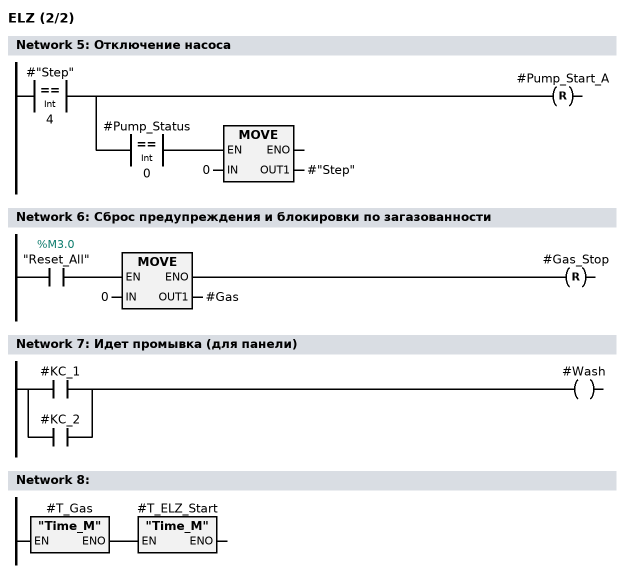
   RUNG wire#powerrail
      { S7_Templates := "SrcType := Int" } EQ_Contact(in1 := #"Step", in2 := 4)
      wire#w1
      R_Coil( #Pump_Start_A )
   END_RUNG
   RUNG wire#w1
      { S7_Templates := "SrcType := Int" } EQ_Contact(in1 := #Pump_Status, in2 := 0)
      Move(in := 0, out1 => #"Step")
   END_RUNG
   // the same network as SCL:
   #_w1 := #"Step" = 4;
   IF #_w1 THEN #Pump_Start_A := FALSE; END_IF;
   IF #_w1 AND (#Pump_Status = 0) THEN #"Step" := 0; END_IF;
END_REGION

REGION Network 6: Сброс предупреждения и блокировки по загазованности
   RUNG wire#powerrail
      Contact( "Reset_All" )
      Move(in := 0, out1 => #Gas)
      R_Coil( #Gas_Stop )
   END_RUNG
   // the same network as SCL:
   IF "Reset_All" THEN
       #Gas := 0;
       #Gas_Stop := FALSE;
   END_IF;
END_REGION

REGION Network 7: Идет промывка (для панели)
   RUNG wire#powerrail
      Contact( #KC_1 )
      wire#w1
      Coil( #Wash )
   END_RUNG
   RUNG wire#powerrail
      Contact( #KC_2 )
   END_RUNG wire#w1
   // the same network as SCL:
   #Wash := #KC_1 OR #KC_2;
END_REGION

REGION Network 8
   RUNG wire#powerrail
      #T_Gas()
      #T_ELZ_Start()
   END_RUNG
   // the same network as SCL:
   #T_Gas(ENO => #_w1);   // "Time_M"
   IF #_w1 THEN
       #T_ELZ_Start();   // "Time_M"
   END_IF;
END_REGION
END_FUNCTION_BLOCK

FUNCTION_BLOCK "Time_M"   // FB92, LAD
{ S7_Optimized_Access := 'FALSE' }
VERSION : 0.1
// stored: AutoNumber false, IsIECCheckEnabled false, SetENOAutomatically false, UDAEnableTagReadback false
   VAR DB_SPECIFIC
      SP_M { S7_SetPoint := 'True'} : Int;
      SP_S { S7_SetPoint := 'True'} : Int := 30;
      Now_M : Int;
      Now_S : Int;
      Rev_M : Int;
      Rev_S : Int;
      Progress : Real;
      Start : Bool;
      "Exit" : Bool;
      Pause : Bool;
      Reset : Bool;
   END_VAR
   VAR_TEMP
      Full_SP_S : Int;
      Full_Now_S : Int;
      Full_Delta_S : Int;
   END_VAR
   VAR_TEMP   // added for the SCL form of the ladder/FBD networks
      _w1 : Bool;
   END_VAR
BEGIN

REGION Network 1: Подсчёт времени
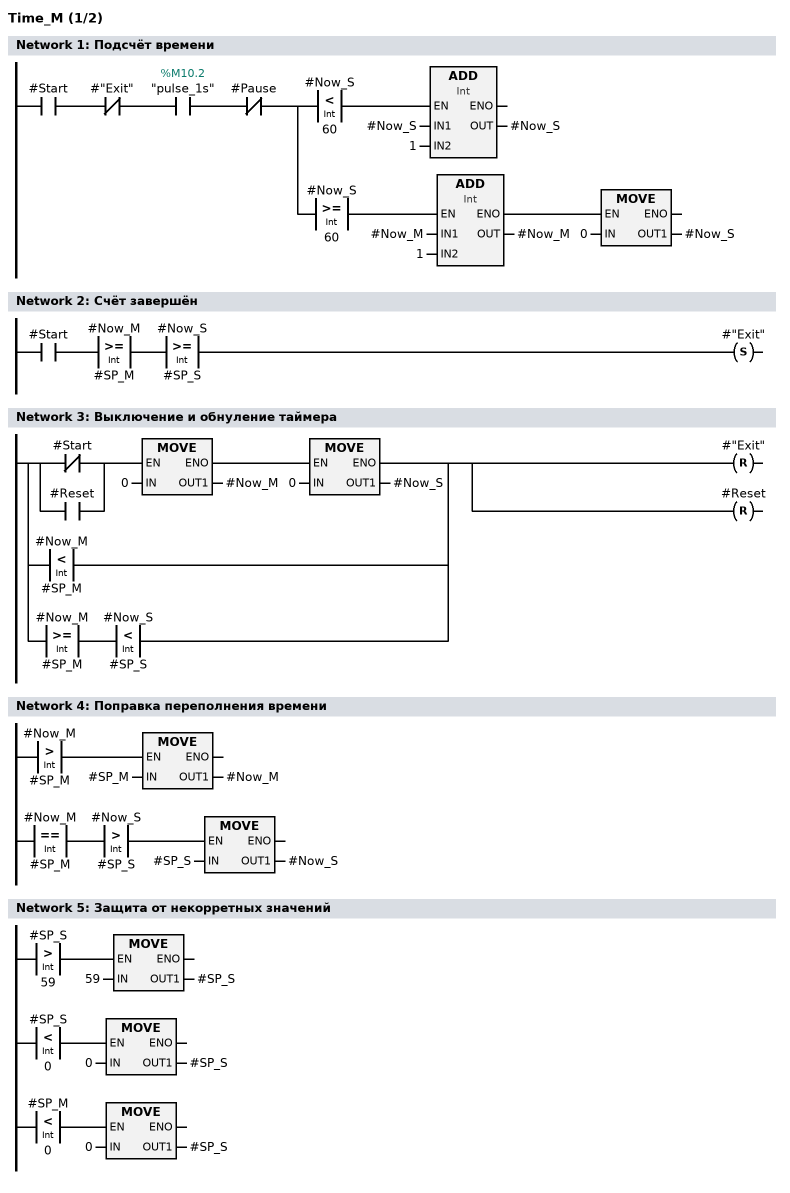
   RUNG wire#powerrail
      Contact( #Start )
      I_Contact( #"Exit" )
      Contact( "pulse_1s" )
      I_Contact( #Pause )
      wire#w1
      { S7_Templates := "SrcType := Int" } LT_Contact(in1 := #Now_S, in2 := 60)
      { S7_Templates := "SrcType := Int"; S7_GenerateENO := "TRUE" } Add(in1 := #Now_S, in2 := 1, out => #Now_S)
   END_RUNG
   RUNG wire#w1
      { S7_Templates := "SrcType := Int" } GE_Contact(in1 := #Now_S, in2 := 60)
      { S7_Templates := "SrcType := Int"; S7_GenerateENO := "TRUE" } Add(in1 := #Now_M, in2 := 1, out => #Now_M)
      { S7_GenerateENO := "TRUE" } Move(in := 0, out1 => #Now_S)
   END_RUNG
   // the same network as SCL:
   // ENO of a box is taken as its EN; it also drops when the box reports an error
   #_w1 := #Start AND NOT #"Exit" AND "pulse_1s" AND NOT #Pause;
   IF #_w1 AND (#Now_S < 60) THEN #Now_S := #Now_S + 1; END_IF;
   IF #_w1 AND (#Now_S >= 60) THEN
       #Now_M := #Now_M + 1;
       #Now_S := 0;
   END_IF;
END_REGION

REGION Network 2: Счёт завершён
   RUNG wire#powerrail
      Contact( #Start )
      { S7_Templates := "SrcType := Int" } GE_Contact(in1 := #Now_M, in2 := #SP_M)
      { S7_Templates := "SrcType := Int" } GE_Contact(in1 := #Now_S, in2 := #SP_S)
      S_Coil( #"Exit" )
   END_RUNG
   // the same network as SCL:
   IF #Start AND (#Now_M >= #SP_M) AND (#Now_S >= #SP_S) THEN #"Exit" := TRUE; END_IF;
END_REGION

REGION Network 3: Выключение и обнуление таймера
   RUNG wire#powerrail
      I_Contact( #Start )
      wire#w1
      { S7_GenerateENO := "TRUE" } Move(in := 0, out1 => #Now_M)
      { S7_GenerateENO := "TRUE" } Move(in := 0, out1 => #Now_S)
      wire#w2
      R_Coil( #"Exit" )
   END_RUNG
   RUNG wire#powerrail
      Contact( #Reset )
   END_RUNG wire#w1
   RUNG wire#powerrail
      { S7_Templates := "SrcType := Int" } LT_Contact(in1 := #Now_M, in2 := #SP_M)
   END_RUNG wire#w2
   RUNG wire#powerrail
      { S7_Templates := "SrcType := Int" } GE_Contact(in1 := #Now_M, in2 := #SP_M)
      { S7_Templates := "SrcType := Int" } LT_Contact(in1 := #Now_S, in2 := #SP_S)
   END_RUNG wire#w2
   RUNG wire#w2
      R_Coil( #Reset )
   END_RUNG
   // the same network as SCL:
   // ENO of a box is taken as its EN; it also drops when the box reports an error
   #_w1 := NOT #Start OR #Reset;
   IF #_w1 THEN
       #Now_M := 0;
       #Now_S := 0;
   END_IF;
   IF #_w1 OR (#Now_M < #SP_M) OR ((#Now_M >= #SP_M) AND (#Now_S < #SP_S)) THEN
       #"Exit" := FALSE;
       #Reset := FALSE;
   END_IF;
END_REGION

REGION Network 4: Поправка переполнения времени
   RUNG wire#powerrail
      { S7_Templates := "SrcType := Int" } GT_Contact(in1 := #Now_M, in2 := #SP_M)
      { S7_GenerateENO := "TRUE" } Move(in := #SP_M, out1 => #Now_M)
   END_RUNG
   RUNG wire#powerrail
      { S7_Templates := "SrcType := Int" } EQ_Contact(in1 := #Now_M, in2 := #SP_M)
      { S7_Templates := "SrcType := Int" } GT_Contact(in1 := #Now_S, in2 := #SP_S)
      { S7_GenerateENO := "TRUE" } Move(in := #SP_S, out1 => #Now_S)
   END_RUNG
   // the same network as SCL:
   IF #Now_M > #SP_M THEN #Now_M := #SP_M; END_IF;
   IF (#Now_M = #SP_M) AND (#Now_S > #SP_S) THEN #Now_S := #SP_S; END_IF;
END_REGION

REGION Network 5: Защита от некорретных значений
   RUNG wire#powerrail
      { S7_Templates := "SrcType := Int" } GT_Contact(in1 := #SP_S, in2 := 59)
      { S7_GenerateENO := "TRUE" } Move(in := 59, out1 => #SP_S)
   END_RUNG
   RUNG wire#powerrail
      { S7_Templates := "SrcType := Int" } LT_Contact(in1 := #SP_S, in2 := 0)
      { S7_GenerateENO := "TRUE" } Move(in := 0, out1 => #SP_S)
   END_RUNG
   RUNG wire#powerrail
      { S7_Templates := "SrcType := Int" } LT_Contact(in1 := #SP_M, in2 := 0)
      { S7_GenerateENO := "TRUE" } Move(in := 0, out1 => #SP_S)
   END_RUNG
   // the same network as SCL:
   IF #SP_S > 59 THEN #SP_S := 59; END_IF;
   IF #SP_S < 0 THEN #SP_S := 0; END_IF;
   IF #SP_M < 0 THEN #SP_S := 0; END_IF;
END_REGION

REGION Network 6: Обратный отсчёт
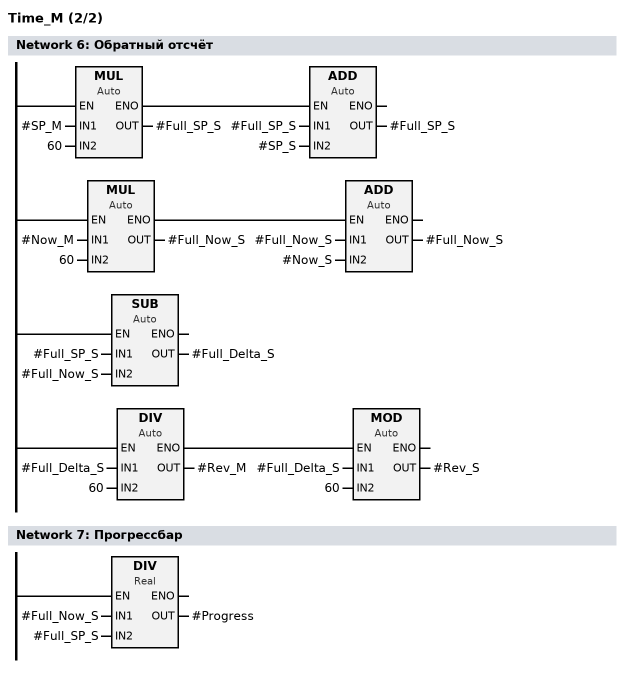
   RUNG wire#powerrail
      Mul(in1 := #SP_M, in2 := 60, out => #Full_SP_S)
      Add(in1 := #Full_SP_S, in2 := #SP_S, out => #Full_SP_S)
   END_RUNG
   RUNG wire#powerrail
      Mul(in1 := #Now_M, in2 := 60, out => #Full_Now_S)
      Add(in1 := #Full_Now_S, in2 := #Now_S, out => #Full_Now_S)
   END_RUNG
   RUNG wire#powerrail
      Sub(in1 := #Full_SP_S, in2 := #Full_Now_S, out => #Full_Delta_S)
   END_RUNG
   RUNG wire#powerrail
      Div(in1 := #Full_Delta_S, in2 := 60, out => #Rev_M)
      Mod(in1 := #Full_Delta_S, in2 := 60, out => #Rev_S)
   END_RUNG
   // the same network as SCL:
   #Full_SP_S := #SP_M * 60;
   #Full_SP_S := #Full_SP_S + #SP_S;
   #Full_Now_S := #Now_M * 60;
   #Full_Now_S := #Full_Now_S + #Now_S;
   #Full_Delta_S := #Full_SP_S - #Full_Now_S;
   #Rev_M := #Full_Delta_S / 60;
   #Rev_S := #Full_Delta_S MOD 60;
END_REGION

REGION Network 7: Прогрессбар
   RUNG wire#powerrail
      { S7_Templates := "SrcType := Real" } Div(in1 := #Full_Now_S, in2 := #Full_SP_S, out => #Progress)
   END_RUNG
   // the same network as SCL:
   #Progress := #Full_Now_S / #Full_SP_S;
END_REGION
END_FUNCTION_BLOCK

FUNCTION_BLOCK "Lock"   // FB2, LAD
{ S7_Optimized_Access := 'TRUE' }
VERSION : 0.1
// stored: AutoNumber true, IsIECCheckEnabled false, IsRetainMemResEnabled false, MemoryReserve 100, SetENOAutomatically false, UDAEnableTagReadback false
BEGIN

REGION Network 1: Блокировка электролизера
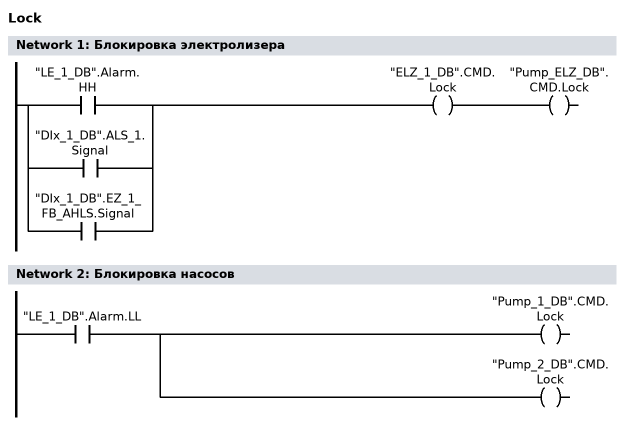
   RUNG wire#powerrail
      Contact( "LE_1_DB".Alarm.HH )
      wire#w1
      Coil( "ELZ_1_DB".CMD.Lock )
      Coil( "Pump_ELZ_DB".CMD.Lock )
   END_RUNG
   RUNG wire#powerrail
      Contact( "DIx_1_DB".ALS_1.Signal )
   END_RUNG wire#w1
   RUNG wire#powerrail
      Contact( "DIx_1_DB".EZ_1_FB_AHLS.Signal )
   END_RUNG wire#w1
   // the same network as SCL:
   "ELZ_1_DB".CMD.Lock := "LE_1_DB".Alarm.HH OR "DIx_1_DB".ALS_1.Signal OR "DIx_1_DB".EZ_1_FB_AHLS.Signal;
   "Pump_ELZ_DB".CMD.Lock := "ELZ_1_DB".CMD.Lock;
END_REGION

REGION Network 2: Блокировка насосов
   RUNG wire#powerrail
      Contact( "LE_1_DB".Alarm.LL )
      wire#w1
      Coil( "Pump_1_DB".CMD.Lock )
   END_RUNG
   RUNG wire#w1
      Coil( "Pump_2_DB".CMD.Lock )
   END_RUNG
   // the same network as SCL:
   "Pump_1_DB".CMD.Lock := "LE_1_DB".Alarm.LL;
   "Pump_2_DB".CMD.Lock := "LE_1_DB".Alarm.LL;
END_REGION
END_FUNCTION_BLOCK

FUNCTION_BLOCK "Line_Control"   // FB5, LAD
{ S7_Optimized_Access := 'FALSE' }
VERSION : 0.1
// stored: AutoNumber false, IsIECCheckEnabled false, SetENOAutomatically false, UDAEnableTagReadback false
   VAR DB_SPECIFIC
      Local : Bool;   // Локальный
      RESET_STAT : Bool;   // Обнуление статистики за неделю
      Line_Settings : Bool;   // Параметры линии
      Line_Alarms : Bool;   // Аварии линии
      Group1_PolyMix_1 : Bool;   // Группа 1 PolyMix 1
      Group1_PolyMix_2 : Bool;   // Группа 1 PolyMix 2
      Group2_PolyMix_1 : Bool;   // Группа 2 PolyMix 1
      Group2_PolyMix_2 : Bool;   // Группа 2 PolyMix 2
      ALLS : Bool;   // Нижний аварийный уровень
      REQ_Z6_BK1 : Bool;   // Запрос открытия задвижки 6 с БК 1
      REQ_Z6_BK2 : Bool;   // Запрос открытия задвижки 6 с БК 2
      REQ_Z5_Start_A : Bool;   // Запрос открытия задвижки 5
      REQ_Z4_Start_A : Bool;   // Запрос открытия задвижки 4
      REQ_Z3_Start_A : Bool;   // Запрос открытия задвижки 3
      REQ_Z2_Start_A : Bool;   // Запрос открытия задвижки 2
      REQ_Z1_Start_A : Bool;   // Запрос открытия задвижки 1
      Line_REQ_Settings : Int;   // Запрос параметров линии
      Line_Now_Settings : Int;   // Параметры линии сейчас
      Line_REQ_Alarms : Int;   // Запрос аварий линии
      Line_Now_Alarms : Int;   // Аварии линии сейчас
      All_Lines : Int := 1;   // Кол-во линий
      All_Pumps : Int := 2;   // Кол-во насосов
      Events : Word;   // События
      pos : Array[0..7] of Bool;   // Вспомогательные переменные
   END_VAR
   VAR
      Line { S7_SetPoint := 'True'} : Array[0..2] of "Block_Line";   // Линии (Block Line)
      Pump { S7_SetPoint := 'True'} : Array[1..2] of "Block_Pump";   // Насосы (Block Pump)
   END_VAR
   VAR DB_SPECIFIC
      Time_DTL : DTL;
   END_VAR
   VAR_TEMP
      summ : Real;
      x1 : Bool;
      x2 : Bool;
   END_VAR
   // Line[1].Flow := 1.0;
   // Line[1].LINE_NUMBER := 1;
   // Line[2].LINE_NUMBER := 2;
   // Line[1..2].Hand := true;
   // Line[0].PID.Settings.Max_out := 1.3;
   // Line[0].PID.Settings.Min_out := 0.7;
   // Line[0].PID.Settings.DeadBand := 0.0;
   // Pump[1].PUMP_NUMBER := 1;
   // Pump[2].PUMP_NUMBER := 2;
   // Pump[1].Line_Main := 1;
   // Pump[2].Line_Main := 2;
   VAR_TEMP   // added for the SCL form of the ladder/FBD networks
      _w1 : Bool;
   END_VAR
BEGIN

REGION Network 1: Вызов функций настроек и аварий линий
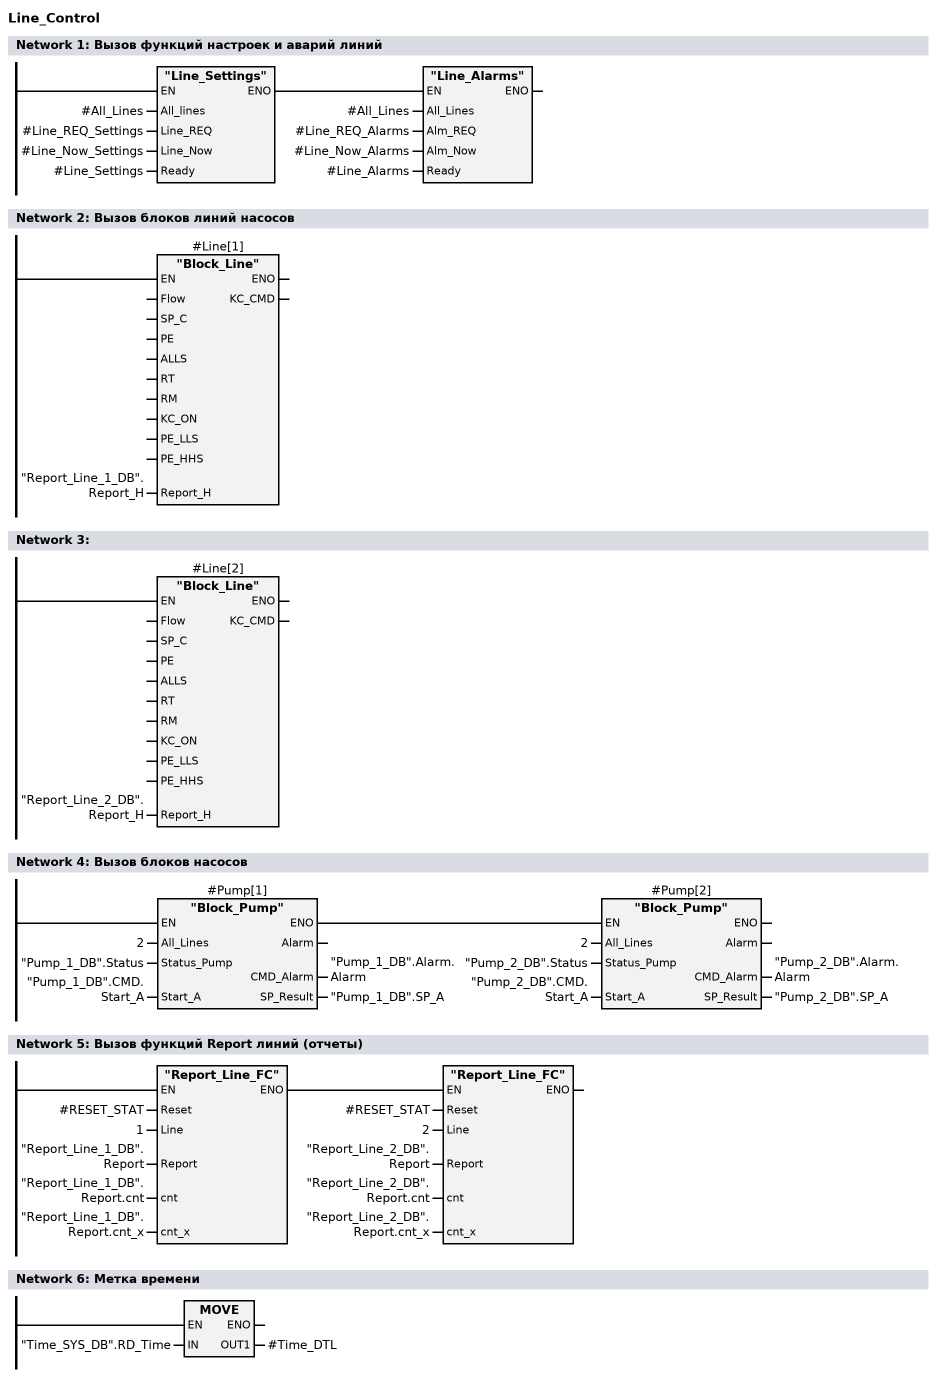
   RUNG wire#powerrail
      "Line_Settings"(All_lines := #All_Lines, Line_REQ := #Line_REQ_Settings, Line_Now := #Line_Now_Settings, Ready := #Line_Settings)
      "Line_Alarms"(All_Lines := #All_Lines, Alm_REQ := #Line_REQ_Alarms, Alm_Now := #Line_Now_Alarms, Ready := #Line_Alarms)
   END_RUNG
   // the same network as SCL:
   "Line_Settings"(All_lines := #All_Lines,
                   Line_REQ := #Line_REQ_Settings,
                   Line_Now := #Line_Now_Settings,
                   Ready := #Line_Settings,
                   ENO => #_w1);
   IF #_w1 THEN
       "Line_Alarms"(All_Lines := #All_Lines,
                     Alm_REQ := #Line_REQ_Alarms,
                     Alm_Now := #Line_Now_Alarms,
                     Ready := #Line_Alarms);
   END_IF;
END_REGION

REGION Network 2: Вызов блоков линий насосов
   RUNG wire#powerrail
      #Line[1](Flow :=, SP_C :=, PE :=, ALLS :=, RT :=, RM :=, KC_ON :=, PE_LLS :=, PE_HHS :=, Report_H := "Report_Line_1_DB".Report_H, KC_CMD =>)
   END_RUNG
   // the same network as SCL:
   #Line[1](Report_H := "Report_Line_1_DB".Report_H);   // "Block_Line"
END_REGION

REGION Network 3
   RUNG wire#powerrail
      #Line[2](Flow :=, SP_C :=, PE :=, ALLS :=, RT :=, RM :=, KC_ON :=, PE_LLS :=, PE_HHS :=, Report_H := "Report_Line_2_DB".Report_H, KC_CMD =>)
   END_RUNG
   // the same network as SCL:
   #Line[2](Report_H := "Report_Line_2_DB".Report_H);   // "Block_Line"
END_REGION

REGION Network 4: Вызов блоков насосов
   RUNG wire#powerrail
      #Pump[1](All_Lines := 2, Status_Pump := "Pump_1_DB".Status, Start_A := "Pump_1_DB".CMD.Start_A, Alarm =>, CMD_Alarm => "Pump_1_DB".Alarm.Alarm, SP_Result => "Pump_1_DB".SP_A)
      #Pump[2](All_Lines := 2, Status_Pump := "Pump_2_DB".Status, Start_A := "Pump_2_DB".CMD.Start_A, Alarm =>, CMD_Alarm => "Pump_2_DB".Alarm.Alarm, SP_Result => "Pump_2_DB".SP_A)
   END_RUNG
   // the same network as SCL:
   #Pump[1](All_Lines := 2,   // "Block_Pump"
            Status_Pump := "Pump_1_DB".Status,
            Start_A := "Pump_1_DB".CMD.Start_A,
            CMD_Alarm => "Pump_1_DB".Alarm.Alarm,
            SP_Result => "Pump_1_DB".SP_A,
            ENO => #_w1);
   IF #_w1 THEN
       #Pump[2](All_Lines := 2,   // "Block_Pump"
                Status_Pump := "Pump_2_DB".Status,
                Start_A := "Pump_2_DB".CMD.Start_A,
                CMD_Alarm => "Pump_2_DB".Alarm.Alarm,
                SP_Result => "Pump_2_DB".SP_A);
   END_IF;
END_REGION

REGION Network 5: Вызов функций Report линий (отчеты)
   RUNG wire#powerrail
      "Report_Line_FC"(Reset := #RESET_STAT, Line := 1, Report := "Report_Line_1_DB".Report, cnt := "Report_Line_1_DB".Report.cnt, cnt_x := "Report_Line_1_DB".Report.cnt_x)
      "Report_Line_FC"(Reset := #RESET_STAT, Line := 2, Report := "Report_Line_2_DB".Report, cnt := "Report_Line_2_DB".Report.cnt, cnt_x := "Report_Line_2_DB".Report.cnt_x)
   END_RUNG
   // the same network as SCL:
   "Report_Line_FC"(Reset := #RESET_STAT,
                    Line := 1,
                    Report := "Report_Line_1_DB".Report,
                    cnt := "Report_Line_1_DB".Report.cnt,
                    cnt_x := "Report_Line_1_DB".Report.cnt_x,
                    ENO => #_w1);
   IF #_w1 THEN
       "Report_Line_FC"(Reset := #RESET_STAT,
                        Line := 2,
                        Report := "Report_Line_2_DB".Report,
                        cnt := "Report_Line_2_DB".Report.cnt,
                        cnt_x := "Report_Line_2_DB".Report.cnt_x);
   END_IF;
END_REGION

REGION Network 6: Метка времени
   RUNG wire#powerrail
      Move(in := "Time_SYS_DB".RD_Time, out1 => #Time_DTL)
   END_RUNG
   // the same network as SCL:
   #Time_DTL := "Time_SYS_DB".RD_Time;
END_REGION
END_FUNCTION_BLOCK

FUNCTION "Line_Settings" : Void   // FC2, LAD
{ S7_Optimized_Access := 'TRUE' }
VERSION : 0.1
// stored: AutoNumber true, IsIECCheckEnabled false, SetENOAutomatically false, UDAEnableTagReadback false
   VAR_INPUT
      All_lines : Int;   // Кол-во линий
   END_VAR
   VAR_IN_OUT
      Line_REQ : Int;   // Запрос линии
      Line_Now : Int;   // Линия сейчас
      Ready : Bool;   // Готовность
   END_VAR
   VAR_TEMP   // added for the SCL form of the ladder/FBD networks
      _w1 : Bool;
      _w2 : Bool;
      _w3 : Bool;
      _w4 : Bool;
      _w5 : Bool;
      _w6 : Bool;
      _w7 : Bool;
      _w8 : Bool;
      _w9 : Bool;
   END_VAR
BEGIN

REGION Network 1: Проверка корректности выбранной линии
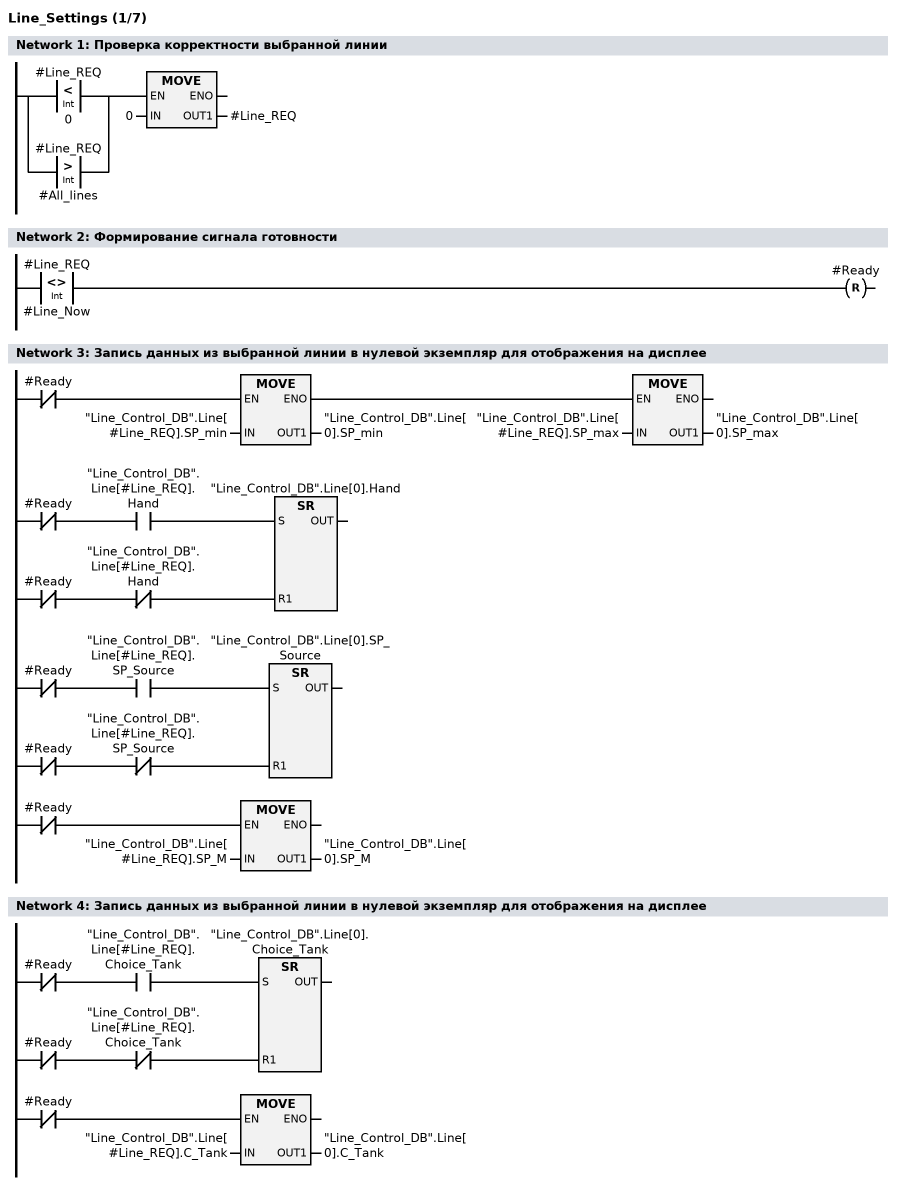
   RUNG wire#powerrail
      { S7_Templates := "SrcType := Int" } LT_Contact(in1 := #Line_REQ, in2 := 0)
      wire#w1
      Move(in := 0, out1 => #Line_REQ)
   END_RUNG
   RUNG wire#powerrail
      { S7_Templates := "SrcType := Int" } GT_Contact(in1 := #Line_REQ, in2 := #All_lines)
   END_RUNG wire#w1
   // the same network as SCL:
   IF (#Line_REQ < 0) OR (#Line_REQ > #All_lines) THEN #Line_REQ := 0; END_IF;
END_REGION

REGION Network 2: Формирование сигнала готовности
   RUNG wire#powerrail
      { S7_Templates := "SrcType := Int" } NE_Contact(in1 := #Line_REQ, in2 := #Line_Now)
      R_Coil( #Ready )
   END_RUNG
   // the same network as SCL:
   IF #Line_REQ <> #Line_Now THEN #Ready := FALSE; END_IF;
END_REGION

REGION Network 3: Запись данных из выбранной линии в нулевой экземпляр для отображения на дисплее
   RUNG wire#powerrail
      I_Contact( #Ready )
      Move(in := "Line_Control_DB".Line[#Line_REQ].SP_min, out1 => "Line_Control_DB".Line[0].SP_min)
      Move(in := "Line_Control_DB".Line[#Line_REQ].SP_max, out1 => "Line_Control_DB".Line[0].SP_max)
   END_RUNG
   RUNG wire#powerrail
      I_Contact( #Ready )
      Contact( "Line_Control_DB".Line[#Line_REQ].Hand )
      S_SR(operand := "Line_Control_DB".Line[0].Hand, r1 := wire#w1)
   END_RUNG
   RUNG wire#powerrail
      I_Contact( #Ready )
      I_Contact( "Line_Control_DB".Line[#Line_REQ].Hand )
   END_RUNG wire#w1
   RUNG wire#powerrail
      I_Contact( #Ready )
      Contact( "Line_Control_DB".Line[#Line_REQ].SP_Source )
      S_SR(operand := "Line_Control_DB".Line[0].SP_Source, r1 := wire#w2)
   END_RUNG
   RUNG wire#powerrail
      I_Contact( #Ready )
      I_Contact( "Line_Control_DB".Line[#Line_REQ].SP_Source )
   END_RUNG wire#w2
   RUNG wire#powerrail
      I_Contact( #Ready )
      Move(in := "Line_Control_DB".Line[#Line_REQ].SP_M, out1 => "Line_Control_DB".Line[0].SP_M)
   END_RUNG
   // the same network as SCL:
   IF NOT #Ready THEN
       "Line_Control_DB".Line[0].SP_min := "Line_Control_DB".Line[#Line_REQ].SP_min;
       "Line_Control_DB".Line[0].SP_max := "Line_Control_DB".Line[#Line_REQ].SP_max;
   END_IF;
   #_w1 := NOT #Ready AND NOT "Line_Control_DB".Line[#Line_REQ].Hand;
   IF NOT #Ready AND "Line_Control_DB".Line[#Line_REQ].Hand THEN
       "Line_Control_DB".Line[0].Hand := TRUE;   // SR flip-flop
   END_IF;
   IF #_w1 THEN "Line_Control_DB".Line[0].Hand := FALSE; END_IF;
   #_w2 := NOT #Ready AND NOT "Line_Control_DB".Line[#Line_REQ].SP_Source;
   IF NOT #Ready AND "Line_Control_DB".Line[#Line_REQ].SP_Source THEN
       "Line_Control_DB".Line[0].SP_Source := TRUE;   // SR flip-flop
   END_IF;
   IF #_w2 THEN "Line_Control_DB".Line[0].SP_Source := FALSE; END_IF;
   IF NOT #Ready THEN "Line_Control_DB".Line[0].SP_M := "Line_Control_DB".Line[#Line_REQ].SP_M; END_IF;
END_REGION

REGION Network 4: Запись данных из выбранной линии в нулевой экземпляр для отображения на дисплее
   RUNG wire#powerrail
      I_Contact( #Ready )
      Contact( "Line_Control_DB".Line[#Line_REQ].Choice_Tank )
      S_SR(operand := "Line_Control_DB".Line[0].Choice_Tank, r1 := wire#w1)
   END_RUNG
   RUNG wire#powerrail
      I_Contact( #Ready )
      I_Contact( "Line_Control_DB".Line[#Line_REQ].Choice_Tank )
   END_RUNG wire#w1
   RUNG wire#powerrail
      I_Contact( #Ready )
      Move(in := "Line_Control_DB".Line[#Line_REQ].C_Tank, out1 => "Line_Control_DB".Line[0].C_Tank)
   END_RUNG
   // the same network as SCL:
   #_w1 := NOT #Ready AND NOT "Line_Control_DB".Line[#Line_REQ].Choice_Tank;
   IF NOT #Ready AND "Line_Control_DB".Line[#Line_REQ].Choice_Tank THEN
       "Line_Control_DB".Line[0].Choice_Tank := TRUE;   // SR flip-flop
   END_IF;
   IF #_w1 THEN "Line_Control_DB".Line[0].Choice_Tank := FALSE; END_IF;
   IF NOT #Ready THEN "Line_Control_DB".Line[0].C_Tank := "Line_Control_DB".Line[#Line_REQ].C_Tank; END_IF;
END_REGION

REGION Network 5: Запись данных из выбранной линии в нулевой экземпляр для отображения на дисплее
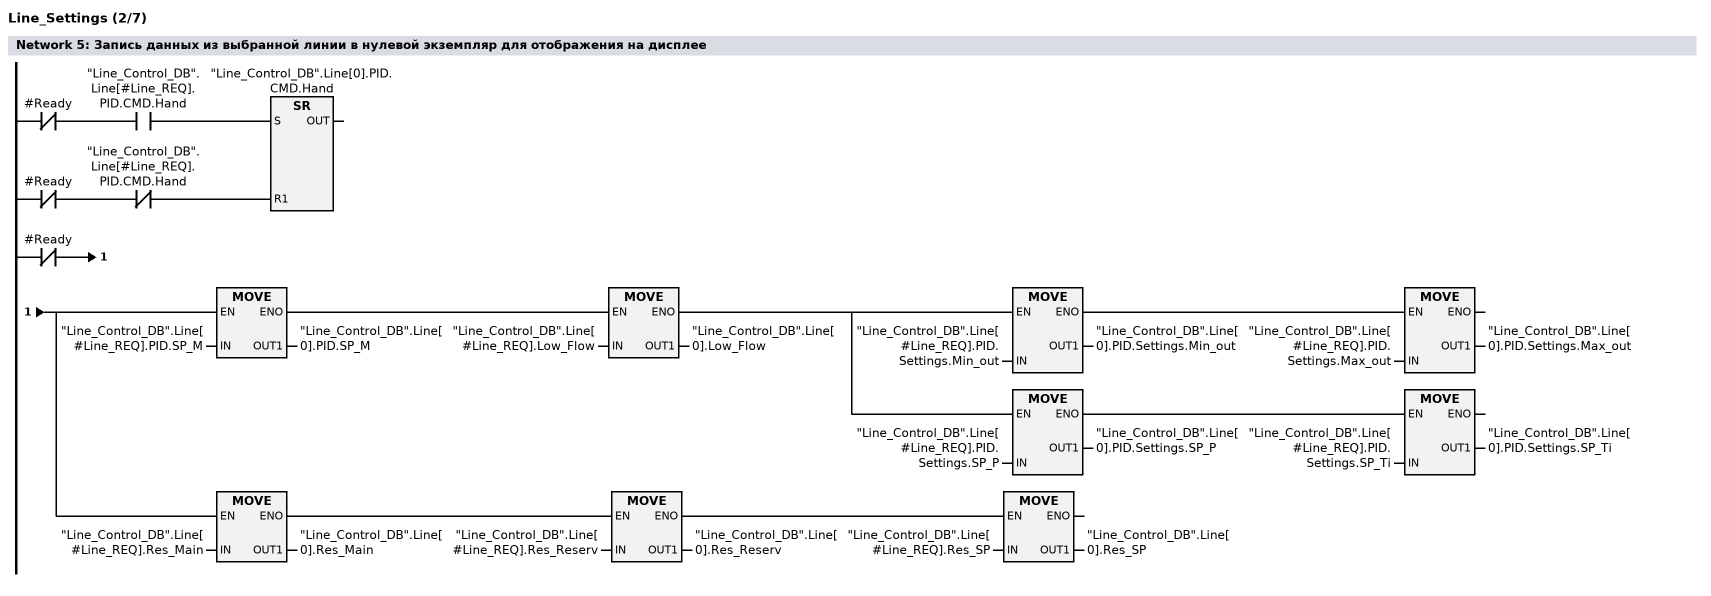
   RUNG wire#powerrail
      I_Contact( #Ready )
      Contact( "Line_Control_DB".Line[#Line_REQ].PID.CMD.Hand )
      S_SR(operand := "Line_Control_DB".Line[0].PID.CMD.Hand, r1 := wire#w1)
   END_RUNG
   RUNG wire#powerrail
      I_Contact( #Ready )
      I_Contact( "Line_Control_DB".Line[#Line_REQ].PID.CMD.Hand )
   END_RUNG wire#w1
   RUNG wire#powerrail
      I_Contact( #Ready )
      wire#w2
      Move(in := "Line_Control_DB".Line[#Line_REQ].PID.SP_M, out1 => "Line_Control_DB".Line[0].PID.SP_M)
      Move(in := "Line_Control_DB".Line[#Line_REQ].Low_Flow, out1 => "Line_Control_DB".Line[0].Low_Flow)
      wire#w3
      Move(in := "Line_Control_DB".Line[#Line_REQ].PID.Settings.Min_out, out1 => "Line_Control_DB".Line[0].PID.Settings.Min_out)
      Move(in := "Line_Control_DB".Line[#Line_REQ].PID.Settings.Max_out, out1 => "Line_Control_DB".Line[0].PID.Settings.Max_out)
   END_RUNG
   RUNG wire#w3
      Move(in := "Line_Control_DB".Line[#Line_REQ].PID.Settings.SP_P, out1 => "Line_Control_DB".Line[0].PID.Settings.SP_P)
      Move(in := "Line_Control_DB".Line[#Line_REQ].PID.Settings.SP_Ti, out1 => "Line_Control_DB".Line[0].PID.Settings.SP_Ti)
   END_RUNG
   RUNG wire#w2
      Move(in := "Line_Control_DB".Line[#Line_REQ].Res_Main, out1 => "Line_Control_DB".Line[0].Res_Main)
      Move(in := "Line_Control_DB".Line[#Line_REQ].Res_Reserv, out1 => "Line_Control_DB".Line[0].Res_Reserv)
      Move(in := "Line_Control_DB".Line[#Line_REQ].Res_SP, out1 => "Line_Control_DB".Line[0].Res_SP)
   END_RUNG
   // the same network as SCL:
   #_w1 := NOT #Ready AND NOT "Line_Control_DB".Line[#Line_REQ].PID.CMD.Hand;
   IF NOT #Ready AND "Line_Control_DB".Line[#Line_REQ].PID.CMD.Hand THEN
       "Line_Control_DB".Line[0].PID.CMD.Hand := TRUE;   // SR flip-flop
   END_IF;
   IF #_w1 THEN "Line_Control_DB".Line[0].PID.CMD.Hand := FALSE; END_IF;
   IF NOT #Ready THEN
       "Line_Control_DB".Line[0].PID.SP_M := "Line_Control_DB".Line[#Line_REQ].PID.SP_M;
       "Line_Control_DB".Line[0].Low_Flow := "Line_Control_DB".Line[#Line_REQ].Low_Flow;
       "Line_Control_DB".Line[0].PID.Settings.Min_out := "Line_Control_DB".Line[#Line_REQ].PID.Settings.Min_out;
       "Line_Control_DB".Line[0].PID.Settings.Max_out := "Line_Control_DB".Line[#Line_REQ].PID.Settings.Max_out;
       "Line_Control_DB".Line[0].PID.Settings.SP_P := "Line_Control_DB".Line[#Line_REQ].PID.Settings.SP_P;
       "Line_Control_DB".Line[0].PID.Settings.SP_Ti := "Line_Control_DB".Line[#Line_REQ].PID.Settings.SP_Ti;
       "Line_Control_DB".Line[0].Res_Main := "Line_Control_DB".Line[#Line_REQ].Res_Main;
       "Line_Control_DB".Line[0].Res_Reserv := "Line_Control_DB".Line[#Line_REQ].Res_Reserv;
       "Line_Control_DB".Line[0].Res_SP := "Line_Control_DB".Line[#Line_REQ].Res_SP;
   END_IF;
END_REGION

REGION Network 6: Запись данных из выбранной линии в нулевой экземпляр для отображения на дисплее
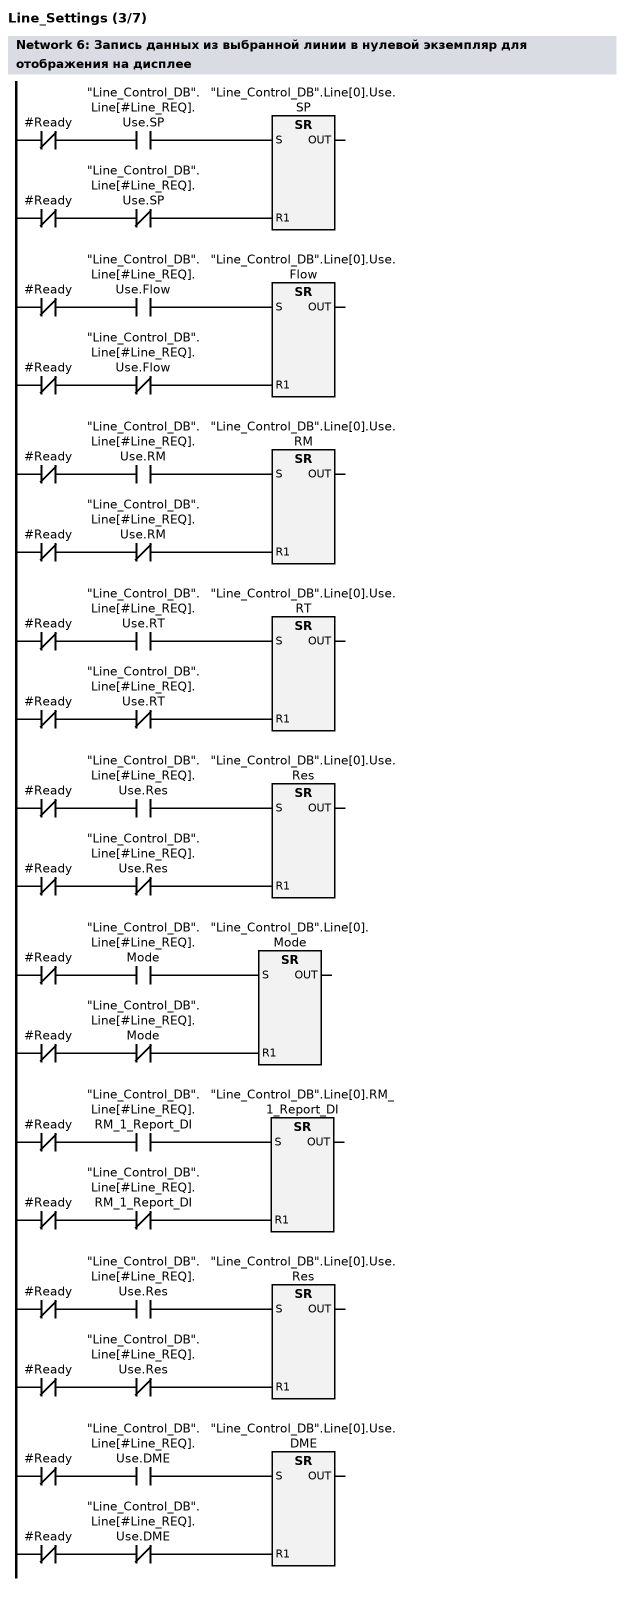
   RUNG wire#powerrail
      I_Contact( #Ready )
      Contact( "Line_Control_DB".Line[#Line_REQ].Use.SP )
      S_SR(operand := "Line_Control_DB".Line[0].Use.SP, r1 := wire#w1)
   END_RUNG
   RUNG wire#powerrail
      I_Contact( #Ready )
      I_Contact( "Line_Control_DB".Line[#Line_REQ].Use.SP )
   END_RUNG wire#w1
   RUNG wire#powerrail
      I_Contact( #Ready )
      Contact( "Line_Control_DB".Line[#Line_REQ].Use.Flow )
      S_SR(operand := "Line_Control_DB".Line[0].Use.Flow, r1 := wire#w2)
   END_RUNG
   RUNG wire#powerrail
      I_Contact( #Ready )
      I_Contact( "Line_Control_DB".Line[#Line_REQ].Use.Flow )
   END_RUNG wire#w2
   RUNG wire#powerrail
      I_Contact( #Ready )
      Contact( "Line_Control_DB".Line[#Line_REQ].Use.RM )
      S_SR(operand := "Line_Control_DB".Line[0].Use.RM, r1 := wire#w3)
   END_RUNG
   RUNG wire#powerrail
      I_Contact( #Ready )
      I_Contact( "Line_Control_DB".Line[#Line_REQ].Use.RM )
   END_RUNG wire#w3
   RUNG wire#powerrail
      I_Contact( #Ready )
      Contact( "Line_Control_DB".Line[#Line_REQ].Use.RT )
      S_SR(operand := "Line_Control_DB".Line[0].Use.RT, r1 := wire#w4)
   END_RUNG
   RUNG wire#powerrail
      I_Contact( #Ready )
      I_Contact( "Line_Control_DB".Line[#Line_REQ].Use.RT )
   END_RUNG wire#w4
   RUNG wire#powerrail
      I_Contact( #Ready )
      Contact( "Line_Control_DB".Line[#Line_REQ].Use.Res )
      S_SR(operand := "Line_Control_DB".Line[0].Use.Res, r1 := wire#w5)
   END_RUNG
   RUNG wire#powerrail
      I_Contact( #Ready )
      I_Contact( "Line_Control_DB".Line[#Line_REQ].Use.Res )
   END_RUNG wire#w5
   RUNG wire#powerrail
      I_Contact( #Ready )
      Contact( "Line_Control_DB".Line[#Line_REQ].Mode )
      S_SR(operand := "Line_Control_DB".Line[0].Mode, r1 := wire#w6)
   END_RUNG
   RUNG wire#powerrail
      I_Contact( #Ready )
      I_Contact( "Line_Control_DB".Line[#Line_REQ].Mode )
   END_RUNG wire#w6
   RUNG wire#powerrail
      I_Contact( #Ready )
      Contact( "Line_Control_DB".Line[#Line_REQ].RM_1_Report_DI )
      S_SR(operand := "Line_Control_DB".Line[0].RM_1_Report_DI, r1 := wire#w7)
   END_RUNG
   RUNG wire#powerrail
      I_Contact( #Ready )
      I_Contact( "Line_Control_DB".Line[#Line_REQ].RM_1_Report_DI )
   END_RUNG wire#w7
   RUNG wire#powerrail
      I_Contact( #Ready )
      Contact( "Line_Control_DB".Line[#Line_REQ].Use.Res )
      S_SR(operand := "Line_Control_DB".Line[0].Use.Res, r1 := wire#w8)
   END_RUNG
   RUNG wire#powerrail
      I_Contact( #Ready )
      I_Contact( "Line_Control_DB".Line[#Line_REQ].Use.Res )
   END_RUNG wire#w8
   RUNG wire#powerrail
      I_Contact( #Ready )
      Contact( "Line_Control_DB".Line[#Line_REQ].Use.DME )
      S_SR(operand := "Line_Control_DB".Line[0].Use.DME, r1 := wire#w9)
   END_RUNG
   RUNG wire#powerrail
      I_Contact( #Ready )
      I_Contact( "Line_Control_DB".Line[#Line_REQ].Use.DME )
   END_RUNG wire#w9
   // the same network as SCL:
   #_w1 := NOT #Ready AND NOT "Line_Control_DB".Line[#Line_REQ].Use.SP;
   IF NOT #Ready AND "Line_Control_DB".Line[#Line_REQ].Use.SP THEN
       "Line_Control_DB".Line[0].Use.SP := TRUE;   // SR flip-flop
   END_IF;
   IF #_w1 THEN "Line_Control_DB".Line[0].Use.SP := FALSE; END_IF;
   #_w2 := NOT #Ready AND NOT "Line_Control_DB".Line[#Line_REQ].Use.Flow;
   IF NOT #Ready AND "Line_Control_DB".Line[#Line_REQ].Use.Flow THEN
       "Line_Control_DB".Line[0].Use.Flow := TRUE;   // SR flip-flop
   END_IF;
   IF #_w2 THEN "Line_Control_DB".Line[0].Use.Flow := FALSE; END_IF;
   #_w3 := NOT #Ready AND NOT "Line_Control_DB".Line[#Line_REQ].Use.RM;
   IF NOT #Ready AND "Line_Control_DB".Line[#Line_REQ].Use.RM THEN
       "Line_Control_DB".Line[0].Use.RM := TRUE;   // SR flip-flop
   END_IF;
   IF #_w3 THEN "Line_Control_DB".Line[0].Use.RM := FALSE; END_IF;
   #_w4 := NOT #Ready AND NOT "Line_Control_DB".Line[#Line_REQ].Use.RT;
   IF NOT #Ready AND "Line_Control_DB".Line[#Line_REQ].Use.RT THEN
       "Line_Control_DB".Line[0].Use.RT := TRUE;   // SR flip-flop
   END_IF;
   IF #_w4 THEN "Line_Control_DB".Line[0].Use.RT := FALSE; END_IF;
   #_w5 := NOT #Ready AND NOT "Line_Control_DB".Line[#Line_REQ].Use.Res;
   IF NOT #Ready AND "Line_Control_DB".Line[#Line_REQ].Use.Res THEN
       "Line_Control_DB".Line[0].Use.Res := TRUE;   // SR flip-flop
   END_IF;
   IF #_w5 THEN "Line_Control_DB".Line[0].Use.Res := FALSE; END_IF;
   #_w6 := NOT #Ready AND NOT "Line_Control_DB".Line[#Line_REQ].Mode;
   IF NOT #Ready AND "Line_Control_DB".Line[#Line_REQ].Mode THEN
       "Line_Control_DB".Line[0].Mode := TRUE;   // SR flip-flop
   END_IF;
   IF #_w6 THEN "Line_Control_DB".Line[0].Mode := FALSE; END_IF;
   #_w7 := NOT #Ready AND NOT "Line_Control_DB".Line[#Line_REQ].RM_1_Report_DI;
   IF NOT #Ready AND "Line_Control_DB".Line[#Line_REQ].RM_1_Report_DI THEN
       "Line_Control_DB".Line[0].RM_1_Report_DI := TRUE;   // SR flip-flop
   END_IF;
   IF #_w7 THEN "Line_Control_DB".Line[0].RM_1_Report_DI := FALSE; END_IF;
   #_w8 := NOT #Ready AND NOT "Line_Control_DB".Line[#Line_REQ].Use.Res;
   IF NOT #Ready AND "Line_Control_DB".Line[#Line_REQ].Use.Res THEN
       "Line_Control_DB".Line[0].Use.Res := TRUE;   // SR flip-flop
   END_IF;
   IF #_w8 THEN "Line_Control_DB".Line[0].Use.Res := FALSE; END_IF;
   #_w9 := NOT #Ready AND NOT "Line_Control_DB".Line[#Line_REQ].Use.DME;
   IF NOT #Ready AND "Line_Control_DB".Line[#Line_REQ].Use.DME THEN
       "Line_Control_DB".Line[0].Use.DME := TRUE;   // SR flip-flop
   END_IF;
   IF #_w9 THEN "Line_Control_DB".Line[0].Use.DME := FALSE; END_IF;
END_REGION

REGION Network 7: Запись данных из выбранной линии в нулевой экземпляр для отображения на дисплее
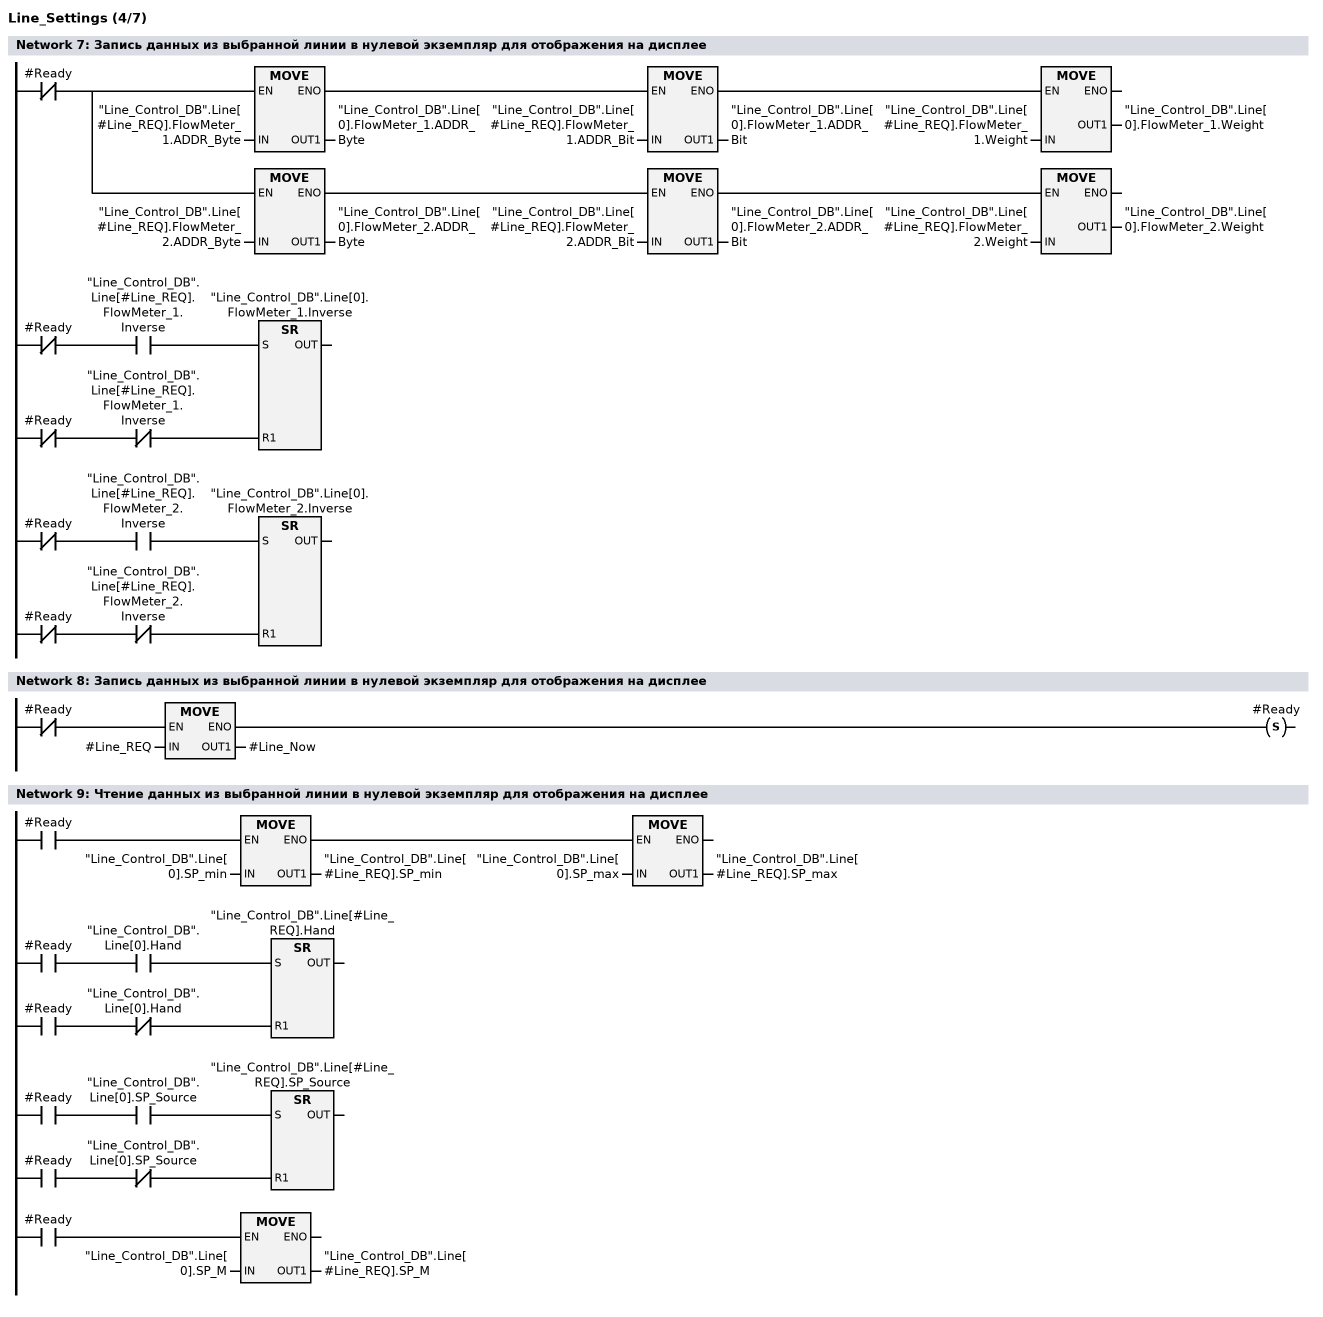
   RUNG wire#powerrail
      I_Contact( #Ready )
      wire#w1
      Move(in := "Line_Control_DB".Line[#Line_REQ].FlowMeter_1.ADDR_Byte, out1 => "Line_Control_DB".Line[0].FlowMeter_1.ADDR_Byte)
      Move(in := "Line_Control_DB".Line[#Line_REQ].FlowMeter_1.ADDR_Bit, out1 => "Line_Control_DB".Line[0].FlowMeter_1.ADDR_Bit)
      Move(in := "Line_Control_DB".Line[#Line_REQ].FlowMeter_1.Weight, out1 => "Line_Control_DB".Line[0].FlowMeter_1.Weight)
   END_RUNG
   RUNG wire#w1
      Move(in := "Line_Control_DB".Line[#Line_REQ].FlowMeter_2.ADDR_Byte, out1 => "Line_Control_DB".Line[0].FlowMeter_2.ADDR_Byte)
      Move(in := "Line_Control_DB".Line[#Line_REQ].FlowMeter_2.ADDR_Bit, out1 => "Line_Control_DB".Line[0].FlowMeter_2.ADDR_Bit)
      Move(in := "Line_Control_DB".Line[#Line_REQ].FlowMeter_2.Weight, out1 => "Line_Control_DB".Line[0].FlowMeter_2.Weight)
   END_RUNG
   RUNG wire#powerrail
      I_Contact( #Ready )
      Contact( "Line_Control_DB".Line[#Line_REQ].FlowMeter_1.Inverse )
      S_SR(operand := "Line_Control_DB".Line[0].FlowMeter_1.Inverse, r1 := wire#w2)
   END_RUNG
   RUNG wire#powerrail
      I_Contact( #Ready )
      I_Contact( "Line_Control_DB".Line[#Line_REQ].FlowMeter_1.Inverse )
   END_RUNG wire#w2
   RUNG wire#powerrail
      I_Contact( #Ready )
      Contact( "Line_Control_DB".Line[#Line_REQ].FlowMeter_2.Inverse )
      S_SR(operand := "Line_Control_DB".Line[0].FlowMeter_2.Inverse, r1 := wire#w3)
   END_RUNG
   RUNG wire#powerrail
      I_Contact( #Ready )
      I_Contact( "Line_Control_DB".Line[#Line_REQ].FlowMeter_2.Inverse )
   END_RUNG wire#w3
   // the same network as SCL:
   IF NOT #Ready THEN
       "Line_Control_DB".Line[0].FlowMeter_1.ADDR_Byte := "Line_Control_DB".Line[#Line_REQ].FlowMeter_1.ADDR_Byte;
       "Line_Control_DB".Line[0].FlowMeter_1.ADDR_Bit := "Line_Control_DB".Line[#Line_REQ].FlowMeter_1.ADDR_Bit;
       "Line_Control_DB".Line[0].FlowMeter_1.Weight := "Line_Control_DB".Line[#Line_REQ].FlowMeter_1.Weight;
       "Line_Control_DB".Line[0].FlowMeter_2.ADDR_Byte := "Line_Control_DB".Line[#Line_REQ].FlowMeter_2.ADDR_Byte;
       "Line_Control_DB".Line[0].FlowMeter_2.ADDR_Bit := "Line_Control_DB".Line[#Line_REQ].FlowMeter_2.ADDR_Bit;
       "Line_Control_DB".Line[0].FlowMeter_2.Weight := "Line_Control_DB".Line[#Line_REQ].FlowMeter_2.Weight;
   END_IF;
   #_w1 := NOT #Ready AND NOT "Line_Control_DB".Line[#Line_REQ].FlowMeter_1.Inverse;
   IF NOT #Ready AND "Line_Control_DB".Line[#Line_REQ].FlowMeter_1.Inverse THEN
       "Line_Control_DB".Line[0].FlowMeter_1.Inverse := TRUE;   // SR flip-flop
   END_IF;
   IF #_w1 THEN "Line_Control_DB".Line[0].FlowMeter_1.Inverse := FALSE; END_IF;
   #_w2 := NOT #Ready AND NOT "Line_Control_DB".Line[#Line_REQ].FlowMeter_2.Inverse;
   IF NOT #Ready AND "Line_Control_DB".Line[#Line_REQ].FlowMeter_2.Inverse THEN
       "Line_Control_DB".Line[0].FlowMeter_2.Inverse := TRUE;   // SR flip-flop
   END_IF;
   IF #_w2 THEN "Line_Control_DB".Line[0].FlowMeter_2.Inverse := FALSE; END_IF;
END_REGION

REGION Network 8: Запись данных из выбранной линии в нулевой экземпляр для отображения на дисплее
   RUNG wire#powerrail
      I_Contact( #Ready )
      Move(in := #Line_REQ, out1 => #Line_Now)
      S_Coil( #Ready )
   END_RUNG
   // the same network as SCL:
   IF NOT #Ready THEN
       #Line_Now := #Line_REQ;
       #Ready := TRUE;
   END_IF;
END_REGION

REGION Network 9: Чтение данных из выбранной линии в нулевой экземпляр для отображения на дисплее
   RUNG wire#powerrail
      Contact( #Ready )
      Move(in := "Line_Control_DB".Line[0].SP_min, out1 => "Line_Control_DB".Line[#Line_REQ].SP_min)
      Move(in := "Line_Control_DB".Line[0].SP_max, out1 => "Line_Control_DB".Line[#Line_REQ].SP_max)
   END_RUNG
   RUNG wire#powerrail
      Contact( #Ready )
      Contact( "Line_Control_DB".Line[0].Hand )
      S_SR(operand := "Line_Control_DB".Line[#Line_REQ].Hand, r1 := wire#w1)
   END_RUNG
   RUNG wire#powerrail
      Contact( #Ready )
      I_Contact( "Line_Control_DB".Line[0].Hand )
   END_RUNG wire#w1
   RUNG wire#powerrail
      Contact( #Ready )
      Contact( "Line_Control_DB".Line[0].SP_Source )
      S_SR(operand := "Line_Control_DB".Line[#Line_REQ].SP_Source, r1 := wire#w2)
   END_RUNG
   RUNG wire#powerrail
      Contact( #Ready )
      I_Contact( "Line_Control_DB".Line[0].SP_Source )
   END_RUNG wire#w2
   RUNG wire#powerrail
      Contact( #Ready )
      Move(in := "Line_Control_DB".Line[0].SP_M, out1 => "Line_Control_DB".Line[#Line_REQ].SP_M)
   END_RUNG
   // the same network as SCL:
   IF #Ready THEN
       "Line_Control_DB".Line[#Line_REQ].SP_min := "Line_Control_DB".Line[0].SP_min;
       "Line_Control_DB".Line[#Line_REQ].SP_max := "Line_Control_DB".Line[0].SP_max;
   END_IF;
   #_w1 := #Ready AND NOT "Line_Control_DB".Line[0].Hand;
   IF #Ready AND "Line_Control_DB".Line[0].Hand THEN
       "Line_Control_DB".Line[#Line_REQ].Hand := TRUE;   // SR flip-flop
   END_IF;
   IF #_w1 THEN "Line_Control_DB".Line[#Line_REQ].Hand := FALSE; END_IF;
   #_w2 := #Ready AND NOT "Line_Control_DB".Line[0].SP_Source;
   IF #Ready AND "Line_Control_DB".Line[0].SP_Source THEN
       "Line_Control_DB".Line[#Line_REQ].SP_Source := TRUE;   // SR flip-flop
   END_IF;
   IF #_w2 THEN "Line_Control_DB".Line[#Line_REQ].SP_Source := FALSE; END_IF;
   IF #Ready THEN "Line_Control_DB".Line[#Line_REQ].SP_M := "Line_Control_DB".Line[0].SP_M; END_IF;
END_REGION

REGION Network 10: Чтение данных из выбранной линии в нулевой экземпляр для отображения на дисплее
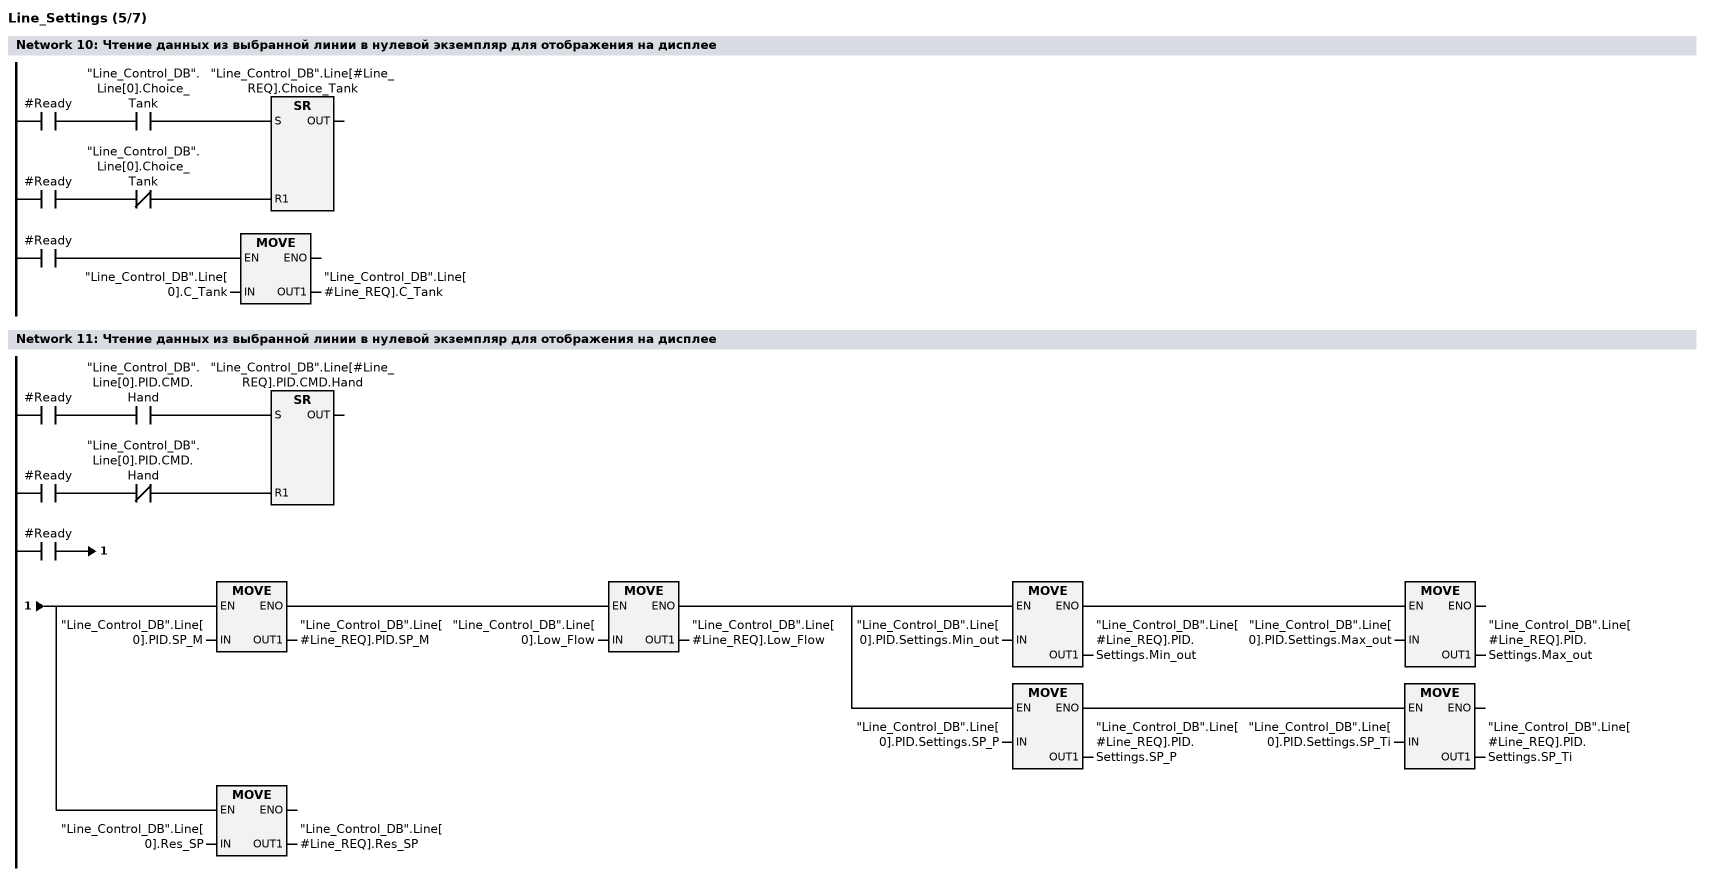
   RUNG wire#powerrail
      Contact( #Ready )
      Contact( "Line_Control_DB".Line[0].Choice_Tank )
      S_SR(operand := "Line_Control_DB".Line[#Line_REQ].Choice_Tank, r1 := wire#w1)
   END_RUNG
   RUNG wire#powerrail
      Contact( #Ready )
      I_Contact( "Line_Control_DB".Line[0].Choice_Tank )
   END_RUNG wire#w1
   RUNG wire#powerrail
      Contact( #Ready )
      Move(in := "Line_Control_DB".Line[0].C_Tank, out1 => "Line_Control_DB".Line[#Line_REQ].C_Tank)
   END_RUNG
   // the same network as SCL:
   #_w1 := #Ready AND NOT "Line_Control_DB".Line[0].Choice_Tank;
   IF #Ready AND "Line_Control_DB".Line[0].Choice_Tank THEN
       "Line_Control_DB".Line[#Line_REQ].Choice_Tank := TRUE;   // SR flip-flop
   END_IF;
   IF #_w1 THEN "Line_Control_DB".Line[#Line_REQ].Choice_Tank := FALSE; END_IF;
   IF #Ready THEN "Line_Control_DB".Line[#Line_REQ].C_Tank := "Line_Control_DB".Line[0].C_Tank; END_IF;
END_REGION

REGION Network 11: Чтение данных из выбранной линии в нулевой экземпляр для отображения на дисплее
   RUNG wire#powerrail
      Contact( #Ready )
      Contact( "Line_Control_DB".Line[0].PID.CMD.Hand )
      S_SR(operand := "Line_Control_DB".Line[#Line_REQ].PID.CMD.Hand, r1 := wire#w1)
   END_RUNG
   RUNG wire#powerrail
      Contact( #Ready )
      I_Contact( "Line_Control_DB".Line[0].PID.CMD.Hand )
   END_RUNG wire#w1
   RUNG wire#powerrail
      Contact( #Ready )
      wire#w2
      Move(in := "Line_Control_DB".Line[0].PID.SP_M, out1 => "Line_Control_DB".Line[#Line_REQ].PID.SP_M)
      Move(in := "Line_Control_DB".Line[0].Low_Flow, out1 => "Line_Control_DB".Line[#Line_REQ].Low_Flow)
      wire#w3
      Move(in := "Line_Control_DB".Line[0].PID.Settings.Min_out, out1 => "Line_Control_DB".Line[#Line_REQ].PID.Settings.Min_out)
      Move(in := "Line_Control_DB".Line[0].PID.Settings.Max_out, out1 => "Line_Control_DB".Line[#Line_REQ].PID.Settings.Max_out)
   END_RUNG
   RUNG wire#w3
      Move(in := "Line_Control_DB".Line[0].PID.Settings.SP_P, out1 => "Line_Control_DB".Line[#Line_REQ].PID.Settings.SP_P)
      Move(in := "Line_Control_DB".Line[0].PID.Settings.SP_Ti, out1 => "Line_Control_DB".Line[#Line_REQ].PID.Settings.SP_Ti)
   END_RUNG
   RUNG wire#w2
      Move(in := "Line_Control_DB".Line[0].Res_SP, out1 => "Line_Control_DB".Line[#Line_REQ].Res_SP)
   END_RUNG
   // the same network as SCL:
   #_w1 := #Ready AND NOT "Line_Control_DB".Line[0].PID.CMD.Hand;
   IF #Ready AND "Line_Control_DB".Line[0].PID.CMD.Hand THEN
       "Line_Control_DB".Line[#Line_REQ].PID.CMD.Hand := TRUE;   // SR flip-flop
   END_IF;
   IF #_w1 THEN "Line_Control_DB".Line[#Line_REQ].PID.CMD.Hand := FALSE; END_IF;
   IF #Ready THEN
       "Line_Control_DB".Line[#Line_REQ].PID.SP_M := "Line_Control_DB".Line[0].PID.SP_M;
       "Line_Control_DB".Line[#Line_REQ].Low_Flow := "Line_Control_DB".Line[0].Low_Flow;
       "Line_Control_DB".Line[#Line_REQ].PID.Settings.Min_out := "Line_Control_DB".Line[0].PID.Settings.Min_out;
       "Line_Control_DB".Line[#Line_REQ].PID.Settings.Max_out := "Line_Control_DB".Line[0].PID.Settings.Max_out;
       "Line_Control_DB".Line[#Line_REQ].PID.Settings.SP_P := "Line_Control_DB".Line[0].PID.Settings.SP_P;
       "Line_Control_DB".Line[#Line_REQ].PID.Settings.SP_Ti := "Line_Control_DB".Line[0].PID.Settings.SP_Ti;
       "Line_Control_DB".Line[#Line_REQ].Res_SP := "Line_Control_DB".Line[0].Res_SP;
   END_IF;
END_REGION

REGION Network 12: Чтение данных из выбранной линии в нулевой экземпляр для отображения на дисплее
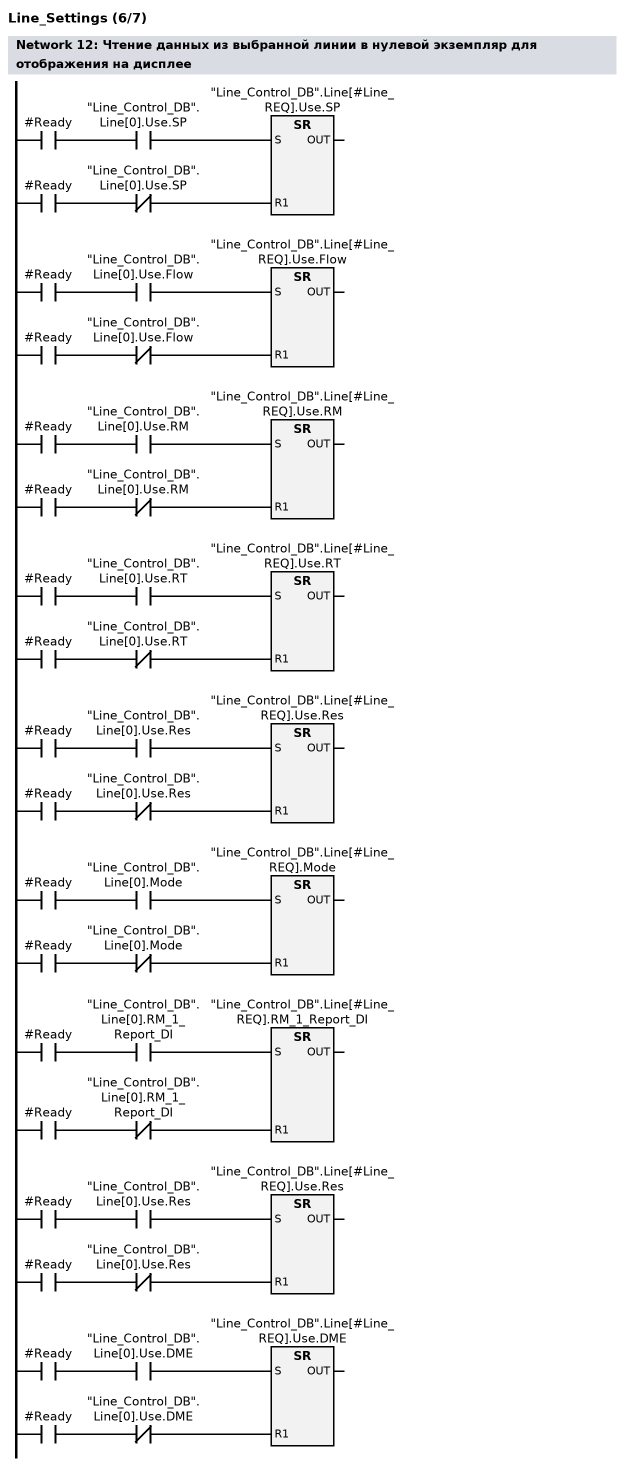
   RUNG wire#powerrail
      Contact( #Ready )
      Contact( "Line_Control_DB".Line[0].Use.SP )
      S_SR(operand := "Line_Control_DB".Line[#Line_REQ].Use.SP, r1 := wire#w1)
   END_RUNG
   RUNG wire#powerrail
      Contact( #Ready )
      I_Contact( "Line_Control_DB".Line[0].Use.SP )
   END_RUNG wire#w1
   RUNG wire#powerrail
      Contact( #Ready )
      Contact( "Line_Control_DB".Line[0].Use.Flow )
      S_SR(operand := "Line_Control_DB".Line[#Line_REQ].Use.Flow, r1 := wire#w2)
   END_RUNG
   RUNG wire#powerrail
      Contact( #Ready )
      I_Contact( "Line_Control_DB".Line[0].Use.Flow )
   END_RUNG wire#w2
   RUNG wire#powerrail
      Contact( #Ready )
      Contact( "Line_Control_DB".Line[0].Use.RM )
      S_SR(operand := "Line_Control_DB".Line[#Line_REQ].Use.RM, r1 := wire#w3)
   END_RUNG
   RUNG wire#powerrail
      Contact( #Ready )
      I_Contact( "Line_Control_DB".Line[0].Use.RM )
   END_RUNG wire#w3
   RUNG wire#powerrail
      Contact( #Ready )
      Contact( "Line_Control_DB".Line[0].Use.RT )
      S_SR(operand := "Line_Control_DB".Line[#Line_REQ].Use.RT, r1 := wire#w4)
   END_RUNG
   RUNG wire#powerrail
      Contact( #Ready )
      I_Contact( "Line_Control_DB".Line[0].Use.RT )
   END_RUNG wire#w4
   RUNG wire#powerrail
      Contact( #Ready )
      Contact( "Line_Control_DB".Line[0].Use.Res )
      S_SR(operand := "Line_Control_DB".Line[#Line_REQ].Use.Res, r1 := wire#w5)
   END_RUNG
   RUNG wire#powerrail
      Contact( #Ready )
      I_Contact( "Line_Control_DB".Line[0].Use.Res )
   END_RUNG wire#w5
   RUNG wire#powerrail
      Contact( #Ready )
      Contact( "Line_Control_DB".Line[0].Mode )
      S_SR(operand := "Line_Control_DB".Line[#Line_REQ].Mode, r1 := wire#w6)
   END_RUNG
   RUNG wire#powerrail
      Contact( #Ready )
      I_Contact( "Line_Control_DB".Line[0].Mode )
   END_RUNG wire#w6
   RUNG wire#powerrail
      Contact( #Ready )
      Contact( "Line_Control_DB".Line[0].RM_1_Report_DI )
      S_SR(operand := "Line_Control_DB".Line[#Line_REQ].RM_1_Report_DI, r1 := wire#w7)
   END_RUNG
   RUNG wire#powerrail
      Contact( #Ready )
      I_Contact( "Line_Control_DB".Line[0].RM_1_Report_DI )
   END_RUNG wire#w7
   RUNG wire#powerrail
      Contact( #Ready )
      Contact( "Line_Control_DB".Line[0].Use.Res )
      S_SR(operand := "Line_Control_DB".Line[#Line_REQ].Use.Res, r1 := wire#w8)
   END_RUNG
   RUNG wire#powerrail
      Contact( #Ready )
      I_Contact( "Line_Control_DB".Line[0].Use.Res )
   END_RUNG wire#w8
   RUNG wire#powerrail
      Contact( #Ready )
      Contact( "Line_Control_DB".Line[0].Use.DME )
      S_SR(operand := "Line_Control_DB".Line[#Line_REQ].Use.DME, r1 := wire#w9)
   END_RUNG
   RUNG wire#powerrail
      Contact( #Ready )
      I_Contact( "Line_Control_DB".Line[0].Use.DME )
   END_RUNG wire#w9
   // the same network as SCL:
   #_w1 := #Ready AND NOT "Line_Control_DB".Line[0].Use.SP;
   IF #Ready AND "Line_Control_DB".Line[0].Use.SP THEN
       "Line_Control_DB".Line[#Line_REQ].Use.SP := TRUE;   // SR flip-flop
   END_IF;
   IF #_w1 THEN "Line_Control_DB".Line[#Line_REQ].Use.SP := FALSE; END_IF;
   #_w2 := #Ready AND NOT "Line_Control_DB".Line[0].Use.Flow;
   IF #Ready AND "Line_Control_DB".Line[0].Use.Flow THEN
       "Line_Control_DB".Line[#Line_REQ].Use.Flow := TRUE;   // SR flip-flop
   END_IF;
   IF #_w2 THEN "Line_Control_DB".Line[#Line_REQ].Use.Flow := FALSE; END_IF;
   #_w3 := #Ready AND NOT "Line_Control_DB".Line[0].Use.RM;
   IF #Ready AND "Line_Control_DB".Line[0].Use.RM THEN
       "Line_Control_DB".Line[#Line_REQ].Use.RM := TRUE;   // SR flip-flop
   END_IF;
   IF #_w3 THEN "Line_Control_DB".Line[#Line_REQ].Use.RM := FALSE; END_IF;
   #_w4 := #Ready AND NOT "Line_Control_DB".Line[0].Use.RT;
   IF #Ready AND "Line_Control_DB".Line[0].Use.RT THEN
       "Line_Control_DB".Line[#Line_REQ].Use.RT := TRUE;   // SR flip-flop
   END_IF;
   IF #_w4 THEN "Line_Control_DB".Line[#Line_REQ].Use.RT := FALSE; END_IF;
   #_w5 := #Ready AND NOT "Line_Control_DB".Line[0].Use.Res;
   IF #Ready AND "Line_Control_DB".Line[0].Use.Res THEN
       "Line_Control_DB".Line[#Line_REQ].Use.Res := TRUE;   // SR flip-flop
   END_IF;
   IF #_w5 THEN "Line_Control_DB".Line[#Line_REQ].Use.Res := FALSE; END_IF;
   #_w6 := #Ready AND NOT "Line_Control_DB".Line[0].Mode;
   IF #Ready AND "Line_Control_DB".Line[0].Mode THEN
       "Line_Control_DB".Line[#Line_REQ].Mode := TRUE;   // SR flip-flop
   END_IF;
   IF #_w6 THEN "Line_Control_DB".Line[#Line_REQ].Mode := FALSE; END_IF;
   #_w7 := #Ready AND NOT "Line_Control_DB".Line[0].RM_1_Report_DI;
   IF #Ready AND "Line_Control_DB".Line[0].RM_1_Report_DI THEN
       "Line_Control_DB".Line[#Line_REQ].RM_1_Report_DI := TRUE;   // SR flip-flop
   END_IF;
   IF #_w7 THEN "Line_Control_DB".Line[#Line_REQ].RM_1_Report_DI := FALSE; END_IF;
   #_w8 := #Ready AND NOT "Line_Control_DB".Line[0].Use.Res;
   IF #Ready AND "Line_Control_DB".Line[0].Use.Res THEN
       "Line_Control_DB".Line[#Line_REQ].Use.Res := TRUE;   // SR flip-flop
   END_IF;
   IF #_w8 THEN "Line_Control_DB".Line[#Line_REQ].Use.Res := FALSE; END_IF;
   #_w9 := #Ready AND NOT "Line_Control_DB".Line[0].Use.DME;
   IF #Ready AND "Line_Control_DB".Line[0].Use.DME THEN
       "Line_Control_DB".Line[#Line_REQ].Use.DME := TRUE;   // SR flip-flop
   END_IF;
   IF #_w9 THEN "Line_Control_DB".Line[#Line_REQ].Use.DME := FALSE; END_IF;
END_REGION

REGION Network 13: Чтение данных из выбранной линии в нулевой экземпляр для отображения на дисплее
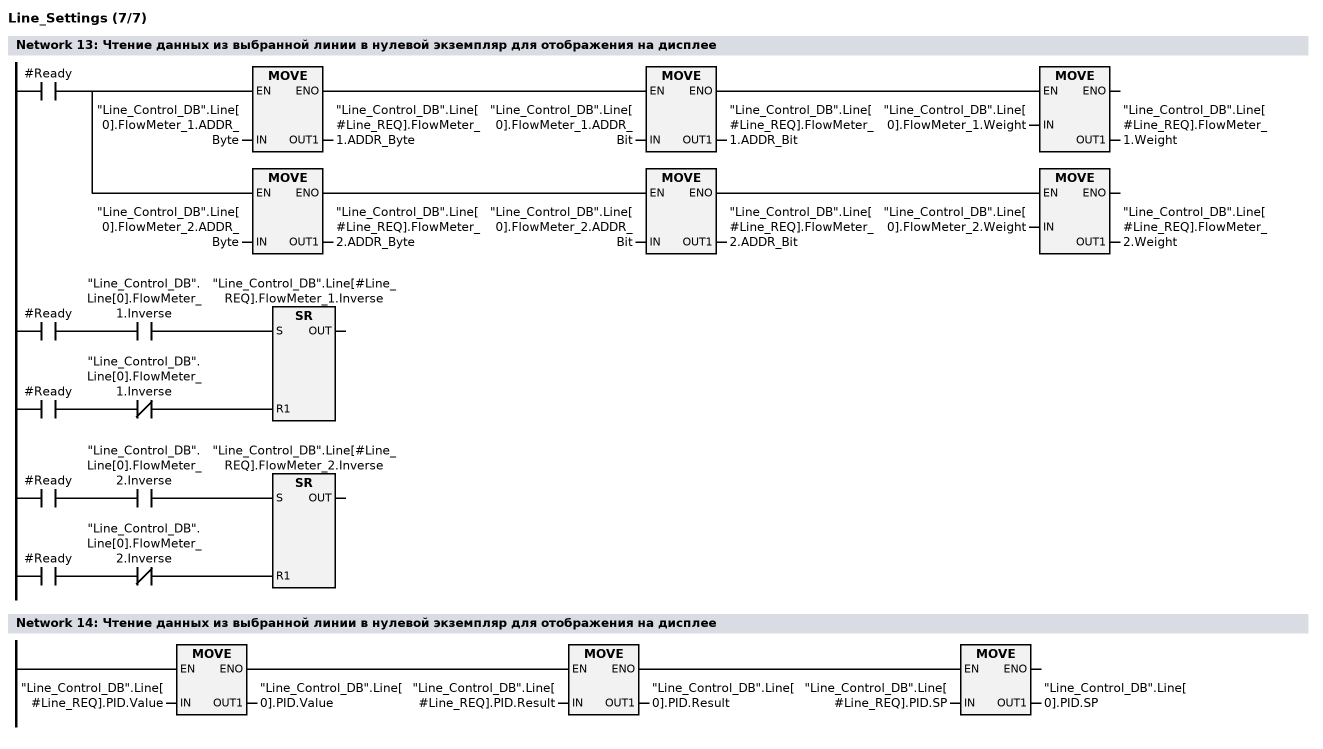
   RUNG wire#powerrail
      Contact( #Ready )
      wire#w1
      Move(in := "Line_Control_DB".Line[0].FlowMeter_1.ADDR_Byte, out1 => "Line_Control_DB".Line[#Line_REQ].FlowMeter_1.ADDR_Byte)
      Move(in := "Line_Control_DB".Line[0].FlowMeter_1.ADDR_Bit, out1 => "Line_Control_DB".Line[#Line_REQ].FlowMeter_1.ADDR_Bit)
      Move(in := "Line_Control_DB".Line[0].FlowMeter_1.Weight, out1 => "Line_Control_DB".Line[#Line_REQ].FlowMeter_1.Weight)
   END_RUNG
   RUNG wire#w1
      Move(in := "Line_Control_DB".Line[0].FlowMeter_2.ADDR_Byte, out1 => "Line_Control_DB".Line[#Line_REQ].FlowMeter_2.ADDR_Byte)
      Move(in := "Line_Control_DB".Line[0].FlowMeter_2.ADDR_Bit, out1 => "Line_Control_DB".Line[#Line_REQ].FlowMeter_2.ADDR_Bit)
      Move(in := "Line_Control_DB".Line[0].FlowMeter_2.Weight, out1 => "Line_Control_DB".Line[#Line_REQ].FlowMeter_2.Weight)
   END_RUNG
   RUNG wire#powerrail
      Contact( #Ready )
      Contact( "Line_Control_DB".Line[0].FlowMeter_1.Inverse )
      S_SR(operand := "Line_Control_DB".Line[#Line_REQ].FlowMeter_1.Inverse, r1 := wire#w2)
   END_RUNG
   RUNG wire#powerrail
      Contact( #Ready )
      I_Contact( "Line_Control_DB".Line[0].FlowMeter_1.Inverse )
   END_RUNG wire#w2
   RUNG wire#powerrail
      Contact( #Ready )
      Contact( "Line_Control_DB".Line[0].FlowMeter_2.Inverse )
      S_SR(operand := "Line_Control_DB".Line[#Line_REQ].FlowMeter_2.Inverse, r1 := wire#w3)
   END_RUNG
   RUNG wire#powerrail
      Contact( #Ready )
      I_Contact( "Line_Control_DB".Line[0].FlowMeter_2.Inverse )
   END_RUNG wire#w3
   // the same network as SCL:
   IF #Ready THEN
       "Line_Control_DB".Line[#Line_REQ].FlowMeter_1.ADDR_Byte := "Line_Control_DB".Line[0].FlowMeter_1.ADDR_Byte;
       "Line_Control_DB".Line[#Line_REQ].FlowMeter_1.ADDR_Bit := "Line_Control_DB".Line[0].FlowMeter_1.ADDR_Bit;
       "Line_Control_DB".Line[#Line_REQ].FlowMeter_1.Weight := "Line_Control_DB".Line[0].FlowMeter_1.Weight;
       "Line_Control_DB".Line[#Line_REQ].FlowMeter_2.ADDR_Byte := "Line_Control_DB".Line[0].FlowMeter_2.ADDR_Byte;
       "Line_Control_DB".Line[#Line_REQ].FlowMeter_2.ADDR_Bit := "Line_Control_DB".Line[0].FlowMeter_2.ADDR_Bit;
       "Line_Control_DB".Line[#Line_REQ].FlowMeter_2.Weight := "Line_Control_DB".Line[0].FlowMeter_2.Weight;
   END_IF;
   #_w1 := #Ready AND NOT "Line_Control_DB".Line[0].FlowMeter_1.Inverse;
   IF #Ready AND "Line_Control_DB".Line[0].FlowMeter_1.Inverse THEN
       "Line_Control_DB".Line[#Line_REQ].FlowMeter_1.Inverse := TRUE;   // SR flip-flop
   END_IF;
   IF #_w1 THEN "Line_Control_DB".Line[#Line_REQ].FlowMeter_1.Inverse := FALSE; END_IF;
   #_w2 := #Ready AND NOT "Line_Control_DB".Line[0].FlowMeter_2.Inverse;
   IF #Ready AND "Line_Control_DB".Line[0].FlowMeter_2.Inverse THEN
       "Line_Control_DB".Line[#Line_REQ].FlowMeter_2.Inverse := TRUE;   // SR flip-flop
   END_IF;
   IF #_w2 THEN "Line_Control_DB".Line[#Line_REQ].FlowMeter_2.Inverse := FALSE; END_IF;
END_REGION

REGION Network 14: Чтение данных из выбранной линии в нулевой экземпляр для отображения на дисплее
   RUNG wire#powerrail
      Move(in := "Line_Control_DB".Line[#Line_REQ].PID.Value, out1 => "Line_Control_DB".Line[0].PID.Value)
      Move(in := "Line_Control_DB".Line[#Line_REQ].PID.Result, out1 => "Line_Control_DB".Line[0].PID.Result)
      Move(in := "Line_Control_DB".Line[#Line_REQ].PID.SP, out1 => "Line_Control_DB".Line[0].PID.SP)
   END_RUNG
   // the same network as SCL:
   "Line_Control_DB".Line[0].PID.Value := "Line_Control_DB".Line[#Line_REQ].PID.Value;
   "Line_Control_DB".Line[0].PID.Result := "Line_Control_DB".Line[#Line_REQ].PID.Result;
   "Line_Control_DB".Line[0].PID.SP := "Line_Control_DB".Line[#Line_REQ].PID.SP;
END_REGION
END_FUNCTION

FUNCTION "Line_Alarms" : Void   // FC3, LAD
{ S7_Optimized_Access := 'TRUE' }
VERSION : 0.1
// stored: AutoNumber true, IsIECCheckEnabled false, SetENOAutomatically false, UDAEnableTagReadback false
   VAR_INPUT
      All_Lines : Int;   // Кол-во линий
   END_VAR
   VAR_IN_OUT
      Alm_REQ : Int;   // Запрос аварии
      Alm_Now : Int;   // Авария сейчас
      Ready : Bool;   // Готовность
   END_VAR
   VAR_TEMP   // added for the SCL form of the ladder/FBD networks
      _w1 : Bool;
      _w2 : Bool;
      _w3 : Bool;
      _w4 : Bool;
      _w5 : Bool;
      _w6 : Bool;
      _w7 : Bool;
   END_VAR
BEGIN

REGION Network 1: Проверка корректности выбранной линии
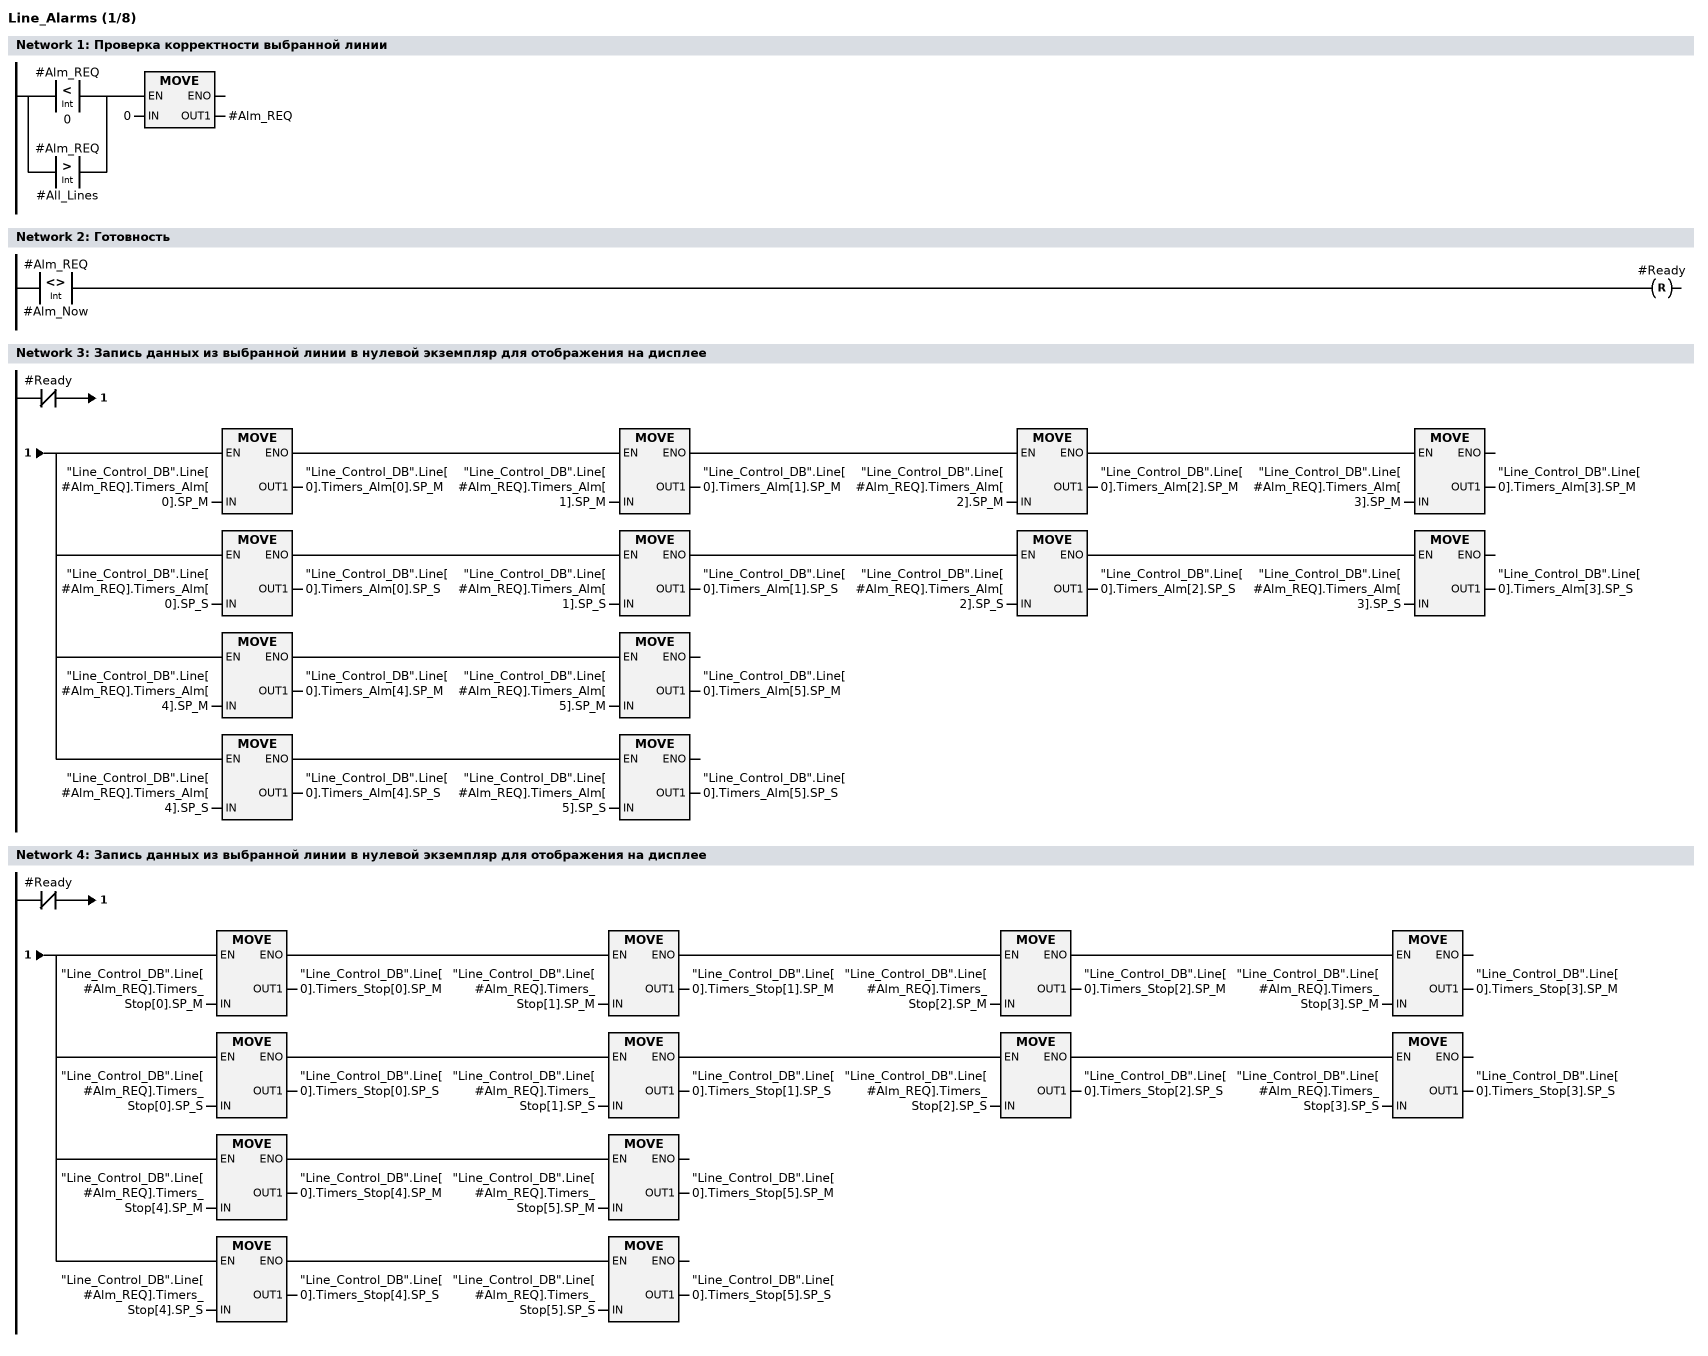
   RUNG wire#powerrail
      { S7_Templates := "SrcType := Int" } LT_Contact(in1 := #Alm_REQ, in2 := 0)
      wire#w1
      Move(in := 0, out1 => #Alm_REQ)
   END_RUNG
   RUNG wire#powerrail
      { S7_Templates := "SrcType := Int" } GT_Contact(in1 := #Alm_REQ, in2 := #All_Lines)
   END_RUNG wire#w1
   // the same network as SCL:
   IF (#Alm_REQ < 0) OR (#Alm_REQ > #All_Lines) THEN #Alm_REQ := 0; END_IF;
END_REGION

REGION Network 2: Готовность
   RUNG wire#powerrail
      { S7_Templates := "SrcType := Int" } NE_Contact(in1 := #Alm_REQ, in2 := #Alm_Now)
      R_Coil( #Ready )
   END_RUNG
   // the same network as SCL:
   IF #Alm_REQ <> #Alm_Now THEN #Ready := FALSE; END_IF;
END_REGION

REGION Network 3: Запись данных из выбранной линии в нулевой экземпляр для отображения на дисплее
   RUNG wire#powerrail
      I_Contact( #Ready )
      wire#w1
      Move(in := "Line_Control_DB".Line[#Alm_REQ].Timers_Alm[0].SP_M, out1 => "Line_Control_DB".Line[0].Timers_Alm[0].SP_M)
      Move(in := "Line_Control_DB".Line[#Alm_REQ].Timers_Alm[1].SP_M, out1 => "Line_Control_DB".Line[0].Timers_Alm[1].SP_M)
      Move(in := "Line_Control_DB".Line[#Alm_REQ].Timers_Alm[2].SP_M, out1 => "Line_Control_DB".Line[0].Timers_Alm[2].SP_M)
      Move(in := "Line_Control_DB".Line[#Alm_REQ].Timers_Alm[3].SP_M, out1 => "Line_Control_DB".Line[0].Timers_Alm[3].SP_M)
   END_RUNG
   RUNG wire#w1
      Move(in := "Line_Control_DB".Line[#Alm_REQ].Timers_Alm[0].SP_S, out1 => "Line_Control_DB".Line[0].Timers_Alm[0].SP_S)
      Move(in := "Line_Control_DB".Line[#Alm_REQ].Timers_Alm[1].SP_S, out1 => "Line_Control_DB".Line[0].Timers_Alm[1].SP_S)
      Move(in := "Line_Control_DB".Line[#Alm_REQ].Timers_Alm[2].SP_S, out1 => "Line_Control_DB".Line[0].Timers_Alm[2].SP_S)
      Move(in := "Line_Control_DB".Line[#Alm_REQ].Timers_Alm[3].SP_S, out1 => "Line_Control_DB".Line[0].Timers_Alm[3].SP_S)
   END_RUNG
   RUNG wire#w1
      Move(in := "Line_Control_DB".Line[#Alm_REQ].Timers_Alm[4].SP_M, out1 => "Line_Control_DB".Line[0].Timers_Alm[4].SP_M)
      Move(in := "Line_Control_DB".Line[#Alm_REQ].Timers_Alm[5].SP_M, out1 => "Line_Control_DB".Line[0].Timers_Alm[5].SP_M)
   END_RUNG
   RUNG wire#w1
      Move(in := "Line_Control_DB".Line[#Alm_REQ].Timers_Alm[4].SP_S, out1 => "Line_Control_DB".Line[0].Timers_Alm[4].SP_S)
      Move(in := "Line_Control_DB".Line[#Alm_REQ].Timers_Alm[5].SP_S, out1 => "Line_Control_DB".Line[0].Timers_Alm[5].SP_S)
   END_RUNG
   // the same network as SCL:
   IF NOT #Ready THEN
       "Line_Control_DB".Line[0].Timers_Alm[0].SP_M := "Line_Control_DB".Line[#Alm_REQ].Timers_Alm[0].SP_M;
       "Line_Control_DB".Line[0].Timers_Alm[1].SP_M := "Line_Control_DB".Line[#Alm_REQ].Timers_Alm[1].SP_M;
       "Line_Control_DB".Line[0].Timers_Alm[2].SP_M := "Line_Control_DB".Line[#Alm_REQ].Timers_Alm[2].SP_M;
       "Line_Control_DB".Line[0].Timers_Alm[3].SP_M := "Line_Control_DB".Line[#Alm_REQ].Timers_Alm[3].SP_M;
       "Line_Control_DB".Line[0].Timers_Alm[0].SP_S := "Line_Control_DB".Line[#Alm_REQ].Timers_Alm[0].SP_S;
       "Line_Control_DB".Line[0].Timers_Alm[1].SP_S := "Line_Control_DB".Line[#Alm_REQ].Timers_Alm[1].SP_S;
       "Line_Control_DB".Line[0].Timers_Alm[2].SP_S := "Line_Control_DB".Line[#Alm_REQ].Timers_Alm[2].SP_S;
       "Line_Control_DB".Line[0].Timers_Alm[3].SP_S := "Line_Control_DB".Line[#Alm_REQ].Timers_Alm[3].SP_S;
       "Line_Control_DB".Line[0].Timers_Alm[4].SP_M := "Line_Control_DB".Line[#Alm_REQ].Timers_Alm[4].SP_M;
       "Line_Control_DB".Line[0].Timers_Alm[5].SP_M := "Line_Control_DB".Line[#Alm_REQ].Timers_Alm[5].SP_M;
       "Line_Control_DB".Line[0].Timers_Alm[4].SP_S := "Line_Control_DB".Line[#Alm_REQ].Timers_Alm[4].SP_S;
       "Line_Control_DB".Line[0].Timers_Alm[5].SP_S := "Line_Control_DB".Line[#Alm_REQ].Timers_Alm[5].SP_S;
   END_IF;
END_REGION

REGION Network 4: Запись данных из выбранной линии в нулевой экземпляр для отображения на дисплее
   RUNG wire#powerrail
      I_Contact( #Ready )
      wire#w1
      Move(in := "Line_Control_DB".Line[#Alm_REQ].Timers_Stop[0].SP_M, out1 => "Line_Control_DB".Line[0].Timers_Stop[0].SP_M)
      Move(in := "Line_Control_DB".Line[#Alm_REQ].Timers_Stop[1].SP_M, out1 => "Line_Control_DB".Line[0].Timers_Stop[1].SP_M)
      Move(in := "Line_Control_DB".Line[#Alm_REQ].Timers_Stop[2].SP_M, out1 => "Line_Control_DB".Line[0].Timers_Stop[2].SP_M)
      Move(in := "Line_Control_DB".Line[#Alm_REQ].Timers_Stop[3].SP_M, out1 => "Line_Control_DB".Line[0].Timers_Stop[3].SP_M)
   END_RUNG
   RUNG wire#w1
      Move(in := "Line_Control_DB".Line[#Alm_REQ].Timers_Stop[0].SP_S, out1 => "Line_Control_DB".Line[0].Timers_Stop[0].SP_S)
      Move(in := "Line_Control_DB".Line[#Alm_REQ].Timers_Stop[1].SP_S, out1 => "Line_Control_DB".Line[0].Timers_Stop[1].SP_S)
      Move(in := "Line_Control_DB".Line[#Alm_REQ].Timers_Stop[2].SP_S, out1 => "Line_Control_DB".Line[0].Timers_Stop[2].SP_S)
      Move(in := "Line_Control_DB".Line[#Alm_REQ].Timers_Stop[3].SP_S, out1 => "Line_Control_DB".Line[0].Timers_Stop[3].SP_S)
   END_RUNG
   RUNG wire#w1
      Move(in := "Line_Control_DB".Line[#Alm_REQ].Timers_Stop[4].SP_M, out1 => "Line_Control_DB".Line[0].Timers_Stop[4].SP_M)
      Move(in := "Line_Control_DB".Line[#Alm_REQ].Timers_Stop[5].SP_M, out1 => "Line_Control_DB".Line[0].Timers_Stop[5].SP_M)
   END_RUNG
   RUNG wire#w1
      Move(in := "Line_Control_DB".Line[#Alm_REQ].Timers_Stop[4].SP_S, out1 => "Line_Control_DB".Line[0].Timers_Stop[4].SP_S)
      Move(in := "Line_Control_DB".Line[#Alm_REQ].Timers_Stop[5].SP_S, out1 => "Line_Control_DB".Line[0].Timers_Stop[5].SP_S)
   END_RUNG
   // the same network as SCL:
   IF NOT #Ready THEN
       "Line_Control_DB".Line[0].Timers_Stop[0].SP_M := "Line_Control_DB".Line[#Alm_REQ].Timers_Stop[0].SP_M;
       "Line_Control_DB".Line[0].Timers_Stop[1].SP_M := "Line_Control_DB".Line[#Alm_REQ].Timers_Stop[1].SP_M;
       "Line_Control_DB".Line[0].Timers_Stop[2].SP_M := "Line_Control_DB".Line[#Alm_REQ].Timers_Stop[2].SP_M;
       "Line_Control_DB".Line[0].Timers_Stop[3].SP_M := "Line_Control_DB".Line[#Alm_REQ].Timers_Stop[3].SP_M;
       "Line_Control_DB".Line[0].Timers_Stop[0].SP_S := "Line_Control_DB".Line[#Alm_REQ].Timers_Stop[0].SP_S;
       "Line_Control_DB".Line[0].Timers_Stop[1].SP_S := "Line_Control_DB".Line[#Alm_REQ].Timers_Stop[1].SP_S;
       "Line_Control_DB".Line[0].Timers_Stop[2].SP_S := "Line_Control_DB".Line[#Alm_REQ].Timers_Stop[2].SP_S;
       "Line_Control_DB".Line[0].Timers_Stop[3].SP_S := "Line_Control_DB".Line[#Alm_REQ].Timers_Stop[3].SP_S;
       "Line_Control_DB".Line[0].Timers_Stop[4].SP_M := "Line_Control_DB".Line[#Alm_REQ].Timers_Stop[4].SP_M;
       "Line_Control_DB".Line[0].Timers_Stop[5].SP_M := "Line_Control_DB".Line[#Alm_REQ].Timers_Stop[5].SP_M;
       "Line_Control_DB".Line[0].Timers_Stop[4].SP_S := "Line_Control_DB".Line[#Alm_REQ].Timers_Stop[4].SP_S;
       "Line_Control_DB".Line[0].Timers_Stop[5].SP_S := "Line_Control_DB".Line[#Alm_REQ].Timers_Stop[5].SP_S;
   END_IF;
END_REGION

REGION Network 5: Запись данных из выбранной линии в нулевой экземпляр для отображения на дисплее
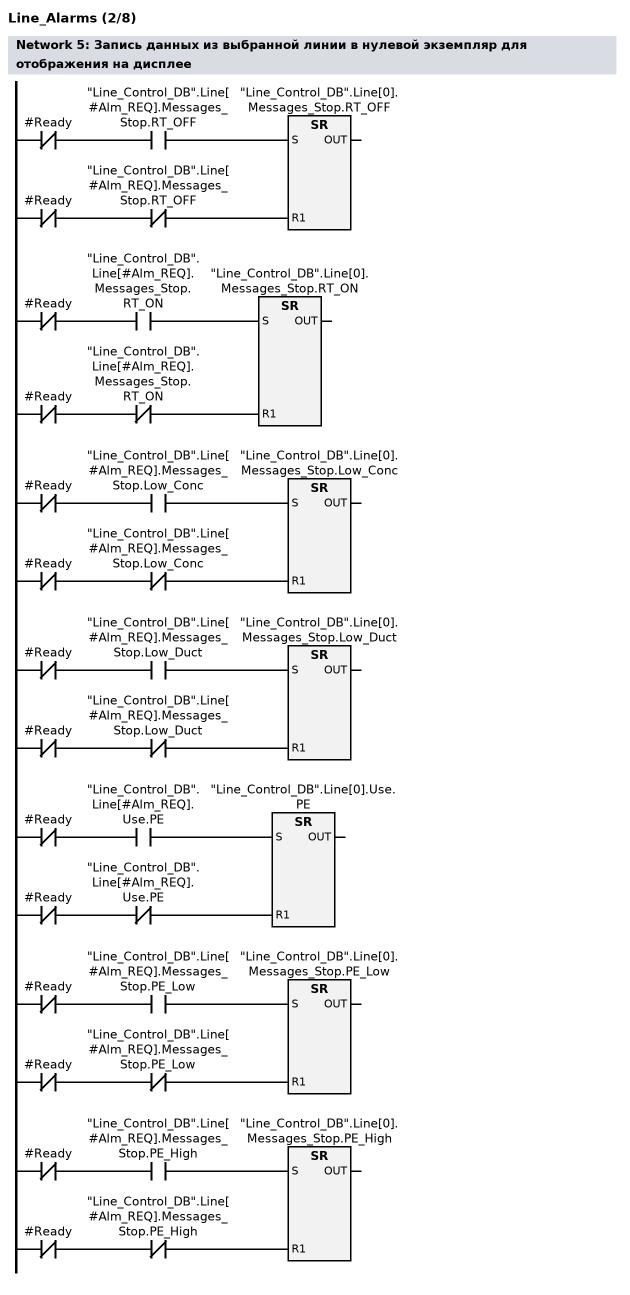
   RUNG wire#powerrail
      I_Contact( #Ready )
      Contact( "Line_Control_DB".Line[#Alm_REQ].Messages_Stop.RT_OFF )
      S_SR(operand := "Line_Control_DB".Line[0].Messages_Stop.RT_OFF, r1 := wire#w1)
   END_RUNG
   RUNG wire#powerrail
      I_Contact( #Ready )
      I_Contact( "Line_Control_DB".Line[#Alm_REQ].Messages_Stop.RT_OFF )
   END_RUNG wire#w1
   RUNG wire#powerrail
      I_Contact( #Ready )
      Contact( "Line_Control_DB".Line[#Alm_REQ].Messages_Stop.RT_ON )
      S_SR(operand := "Line_Control_DB".Line[0].Messages_Stop.RT_ON, r1 := wire#w2)
   END_RUNG
   RUNG wire#powerrail
      I_Contact( #Ready )
      I_Contact( "Line_Control_DB".Line[#Alm_REQ].Messages_Stop.RT_ON )
   END_RUNG wire#w2
   RUNG wire#powerrail
      I_Contact( #Ready )
      Contact( "Line_Control_DB".Line[#Alm_REQ].Messages_Stop.Low_Conc )
      S_SR(operand := "Line_Control_DB".Line[0].Messages_Stop.Low_Conc, r1 := wire#w3)
   END_RUNG
   RUNG wire#powerrail
      I_Contact( #Ready )
      I_Contact( "Line_Control_DB".Line[#Alm_REQ].Messages_Stop.Low_Conc )
   END_RUNG wire#w3
   RUNG wire#powerrail
      I_Contact( #Ready )
      Contact( "Line_Control_DB".Line[#Alm_REQ].Messages_Stop.Low_Duct )
      S_SR(operand := "Line_Control_DB".Line[0].Messages_Stop.Low_Duct, r1 := wire#w4)
   END_RUNG
   RUNG wire#powerrail
      I_Contact( #Ready )
      I_Contact( "Line_Control_DB".Line[#Alm_REQ].Messages_Stop.Low_Duct )
   END_RUNG wire#w4
   RUNG wire#powerrail
      I_Contact( #Ready )
      Contact( "Line_Control_DB".Line[#Alm_REQ].Use.PE )
      S_SR(operand := "Line_Control_DB".Line[0].Use.PE, r1 := wire#w5)
   END_RUNG
   RUNG wire#powerrail
      I_Contact( #Ready )
      I_Contact( "Line_Control_DB".Line[#Alm_REQ].Use.PE )
   END_RUNG wire#w5
   RUNG wire#powerrail
      I_Contact( #Ready )
      Contact( "Line_Control_DB".Line[#Alm_REQ].Messages_Stop.PE_Low )
      S_SR(operand := "Line_Control_DB".Line[0].Messages_Stop.PE_Low, r1 := wire#w6)
   END_RUNG
   RUNG wire#powerrail
      I_Contact( #Ready )
      I_Contact( "Line_Control_DB".Line[#Alm_REQ].Messages_Stop.PE_Low )
   END_RUNG wire#w6
   RUNG wire#powerrail
      I_Contact( #Ready )
      Contact( "Line_Control_DB".Line[#Alm_REQ].Messages_Stop.PE_High )
      S_SR(operand := "Line_Control_DB".Line[0].Messages_Stop.PE_High, r1 := wire#w7)
   END_RUNG
   RUNG wire#powerrail
      I_Contact( #Ready )
      I_Contact( "Line_Control_DB".Line[#Alm_REQ].Messages_Stop.PE_High )
   END_RUNG wire#w7
   // the same network as SCL:
   #_w1 := NOT #Ready AND NOT "Line_Control_DB".Line[#Alm_REQ].Messages_Stop.RT_OFF;
   IF NOT #Ready AND "Line_Control_DB".Line[#Alm_REQ].Messages_Stop.RT_OFF THEN
       "Line_Control_DB".Line[0].Messages_Stop.RT_OFF := TRUE;   // SR flip-flop
   END_IF;
   IF #_w1 THEN "Line_Control_DB".Line[0].Messages_Stop.RT_OFF := FALSE; END_IF;
   #_w2 := NOT #Ready AND NOT "Line_Control_DB".Line[#Alm_REQ].Messages_Stop.RT_ON;
   IF NOT #Ready AND "Line_Control_DB".Line[#Alm_REQ].Messages_Stop.RT_ON THEN
       "Line_Control_DB".Line[0].Messages_Stop.RT_ON := TRUE;   // SR flip-flop
   END_IF;
   IF #_w2 THEN "Line_Control_DB".Line[0].Messages_Stop.RT_ON := FALSE; END_IF;
   #_w3 := NOT #Ready AND NOT "Line_Control_DB".Line[#Alm_REQ].Messages_Stop.Low_Conc;
   IF NOT #Ready AND "Line_Control_DB".Line[#Alm_REQ].Messages_Stop.Low_Conc THEN
       "Line_Control_DB".Line[0].Messages_Stop.Low_Conc := TRUE;   // SR flip-flop
   END_IF;
   IF #_w3 THEN "Line_Control_DB".Line[0].Messages_Stop.Low_Conc := FALSE; END_IF;
   #_w4 := NOT #Ready AND NOT "Line_Control_DB".Line[#Alm_REQ].Messages_Stop.Low_Duct;
   IF NOT #Ready AND "Line_Control_DB".Line[#Alm_REQ].Messages_Stop.Low_Duct THEN
       "Line_Control_DB".Line[0].Messages_Stop.Low_Duct := TRUE;   // SR flip-flop
   END_IF;
   IF #_w4 THEN "Line_Control_DB".Line[0].Messages_Stop.Low_Duct := FALSE; END_IF;
   #_w5 := NOT #Ready AND NOT "Line_Control_DB".Line[#Alm_REQ].Use.PE;
   IF NOT #Ready AND "Line_Control_DB".Line[#Alm_REQ].Use.PE THEN
       "Line_Control_DB".Line[0].Use.PE := TRUE;   // SR flip-flop
   END_IF;
   IF #_w5 THEN "Line_Control_DB".Line[0].Use.PE := FALSE; END_IF;
   #_w6 := NOT #Ready AND NOT "Line_Control_DB".Line[#Alm_REQ].Messages_Stop.PE_Low;
   IF NOT #Ready AND "Line_Control_DB".Line[#Alm_REQ].Messages_Stop.PE_Low THEN
       "Line_Control_DB".Line[0].Messages_Stop.PE_Low := TRUE;   // SR flip-flop
   END_IF;
   IF #_w6 THEN "Line_Control_DB".Line[0].Messages_Stop.PE_Low := FALSE; END_IF;
   #_w7 := NOT #Ready AND NOT "Line_Control_DB".Line[#Alm_REQ].Messages_Stop.PE_High;
   IF NOT #Ready AND "Line_Control_DB".Line[#Alm_REQ].Messages_Stop.PE_High THEN
       "Line_Control_DB".Line[0].Messages_Stop.PE_High := TRUE;   // SR flip-flop
   END_IF;
   IF #_w7 THEN "Line_Control_DB".Line[0].Messages_Stop.PE_High := FALSE; END_IF;
END_REGION

REGION Network 6: Запись данных из выбранной линии в нулевой экземпляр для отображения на дисплее
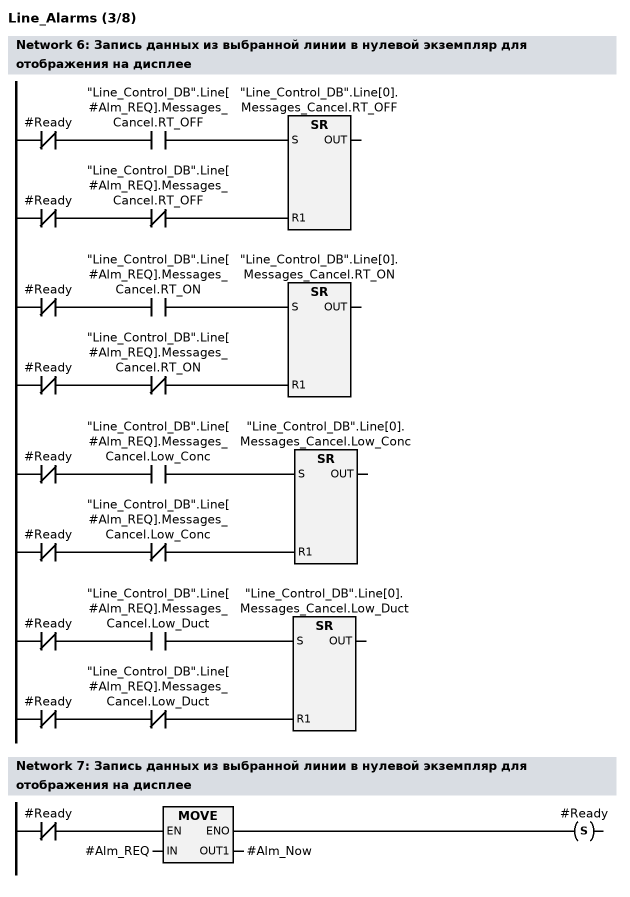
   RUNG wire#powerrail
      I_Contact( #Ready )
      Contact( "Line_Control_DB".Line[#Alm_REQ].Messages_Cancel.RT_OFF )
      S_SR(operand := "Line_Control_DB".Line[0].Messages_Cancel.RT_OFF, r1 := wire#w1)
   END_RUNG
   RUNG wire#powerrail
      I_Contact( #Ready )
      I_Contact( "Line_Control_DB".Line[#Alm_REQ].Messages_Cancel.RT_OFF )
   END_RUNG wire#w1
   RUNG wire#powerrail
      I_Contact( #Ready )
      Contact( "Line_Control_DB".Line[#Alm_REQ].Messages_Cancel.RT_ON )
      S_SR(operand := "Line_Control_DB".Line[0].Messages_Cancel.RT_ON, r1 := wire#w2)
   END_RUNG
   RUNG wire#powerrail
      I_Contact( #Ready )
      I_Contact( "Line_Control_DB".Line[#Alm_REQ].Messages_Cancel.RT_ON )
   END_RUNG wire#w2
   RUNG wire#powerrail
      I_Contact( #Ready )
      Contact( "Line_Control_DB".Line[#Alm_REQ].Messages_Cancel.Low_Conc )
      S_SR(operand := "Line_Control_DB".Line[0].Messages_Cancel.Low_Conc, r1 := wire#w3)
   END_RUNG
   RUNG wire#powerrail
      I_Contact( #Ready )
      I_Contact( "Line_Control_DB".Line[#Alm_REQ].Messages_Cancel.Low_Conc )
   END_RUNG wire#w3
   RUNG wire#powerrail
      I_Contact( #Ready )
      Contact( "Line_Control_DB".Line[#Alm_REQ].Messages_Cancel.Low_Duct )
      S_SR(operand := "Line_Control_DB".Line[0].Messages_Cancel.Low_Duct, r1 := wire#w4)
   END_RUNG
   RUNG wire#powerrail
      I_Contact( #Ready )
      I_Contact( "Line_Control_DB".Line[#Alm_REQ].Messages_Cancel.Low_Duct )
   END_RUNG wire#w4
   // the same network as SCL:
   #_w1 := NOT #Ready AND NOT "Line_Control_DB".Line[#Alm_REQ].Messages_Cancel.RT_OFF;
   IF NOT #Ready AND "Line_Control_DB".Line[#Alm_REQ].Messages_Cancel.RT_OFF THEN
       "Line_Control_DB".Line[0].Messages_Cancel.RT_OFF := TRUE;   // SR flip-flop
   END_IF;
   IF #_w1 THEN "Line_Control_DB".Line[0].Messages_Cancel.RT_OFF := FALSE; END_IF;
   #_w2 := NOT #Ready AND NOT "Line_Control_DB".Line[#Alm_REQ].Messages_Cancel.RT_ON;
   IF NOT #Ready AND "Line_Control_DB".Line[#Alm_REQ].Messages_Cancel.RT_ON THEN
       "Line_Control_DB".Line[0].Messages_Cancel.RT_ON := TRUE;   // SR flip-flop
   END_IF;
   IF #_w2 THEN "Line_Control_DB".Line[0].Messages_Cancel.RT_ON := FALSE; END_IF;
   #_w3 := NOT #Ready AND NOT "Line_Control_DB".Line[#Alm_REQ].Messages_Cancel.Low_Conc;
   IF NOT #Ready AND "Line_Control_DB".Line[#Alm_REQ].Messages_Cancel.Low_Conc THEN
       "Line_Control_DB".Line[0].Messages_Cancel.Low_Conc := TRUE;   // SR flip-flop
   END_IF;
   IF #_w3 THEN "Line_Control_DB".Line[0].Messages_Cancel.Low_Conc := FALSE; END_IF;
   #_w4 := NOT #Ready AND NOT "Line_Control_DB".Line[#Alm_REQ].Messages_Cancel.Low_Duct;
   IF NOT #Ready AND "Line_Control_DB".Line[#Alm_REQ].Messages_Cancel.Low_Duct THEN
       "Line_Control_DB".Line[0].Messages_Cancel.Low_Duct := TRUE;   // SR flip-flop
   END_IF;
   IF #_w4 THEN "Line_Control_DB".Line[0].Messages_Cancel.Low_Duct := FALSE; END_IF;
END_REGION

REGION Network 7: Запись данных из выбранной линии в нулевой экземпляр для отображения на дисплее
   RUNG wire#powerrail
      I_Contact( #Ready )
      Move(in := #Alm_REQ, out1 => #Alm_Now)
      S_Coil( #Ready )
   END_RUNG
   // the same network as SCL:
   IF NOT #Ready THEN
       #Alm_Now := #Alm_REQ;
       #Ready := TRUE;
   END_IF;
END_REGION

REGION Network 8: Запись данных из выбранной линии в нулевой экземпляр для отображения на дисплее
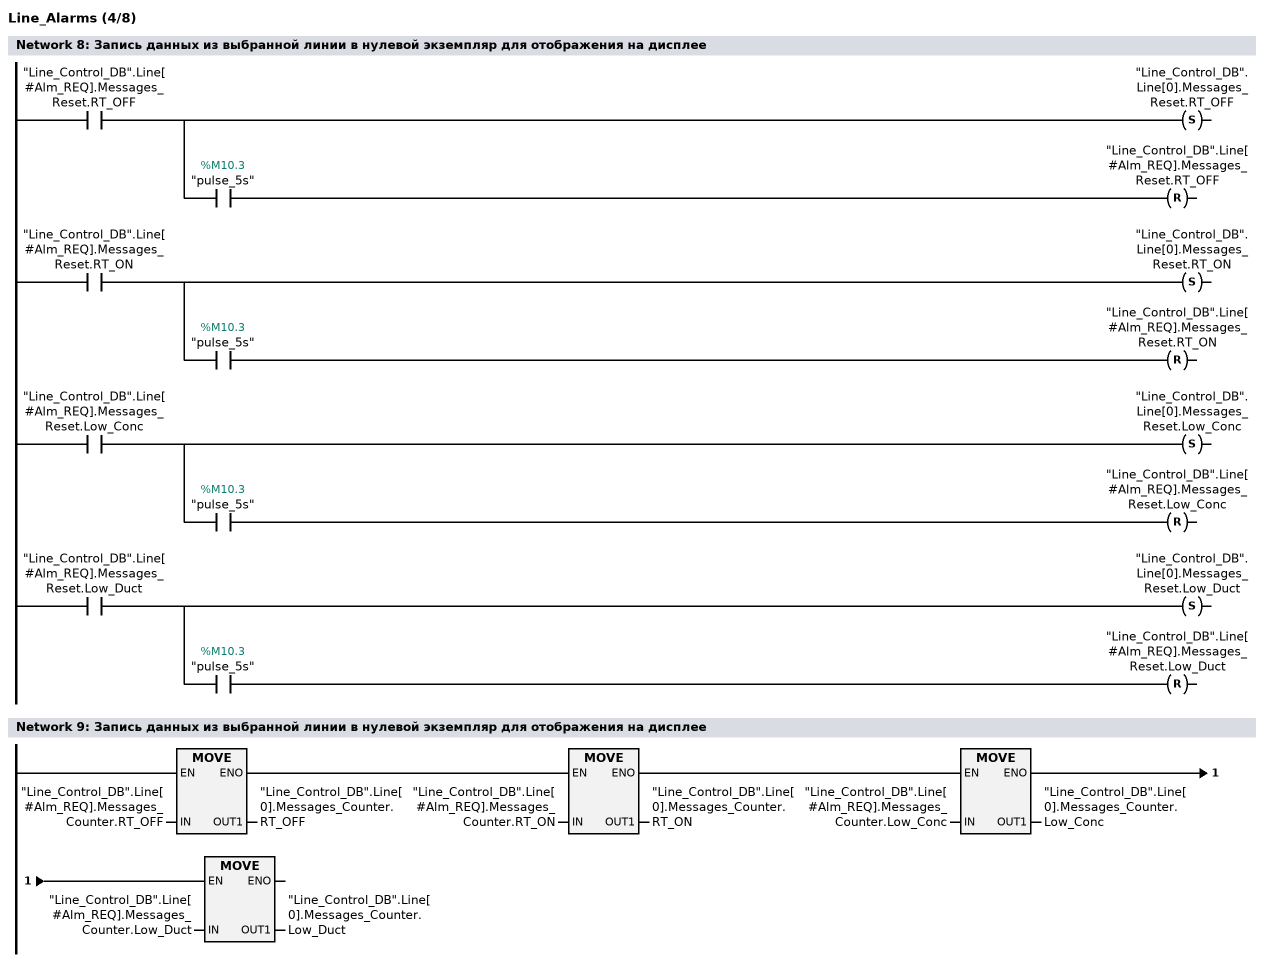
   RUNG wire#powerrail
      Contact( "Line_Control_DB".Line[#Alm_REQ].Messages_Reset.RT_OFF )
      wire#w1
      S_Coil( "Line_Control_DB".Line[0].Messages_Reset.RT_OFF )
   END_RUNG
   RUNG wire#w1
      Contact( "pulse_5s" )
      R_Coil( "Line_Control_DB".Line[#Alm_REQ].Messages_Reset.RT_OFF )
   END_RUNG
   RUNG wire#powerrail
      Contact( "Line_Control_DB".Line[#Alm_REQ].Messages_Reset.RT_ON )
      wire#w2
      S_Coil( "Line_Control_DB".Line[0].Messages_Reset.RT_ON )
   END_RUNG
   RUNG wire#w2
      Contact( "pulse_5s" )
      R_Coil( "Line_Control_DB".Line[#Alm_REQ].Messages_Reset.RT_ON )
   END_RUNG
   RUNG wire#powerrail
      Contact( "Line_Control_DB".Line[#Alm_REQ].Messages_Reset.Low_Conc )
      wire#w3
      S_Coil( "Line_Control_DB".Line[0].Messages_Reset.Low_Conc )
   END_RUNG
   RUNG wire#w3
      Contact( "pulse_5s" )
      R_Coil( "Line_Control_DB".Line[#Alm_REQ].Messages_Reset.Low_Conc )
   END_RUNG
   RUNG wire#powerrail
      Contact( "Line_Control_DB".Line[#Alm_REQ].Messages_Reset.Low_Duct )
      wire#w4
      S_Coil( "Line_Control_DB".Line[0].Messages_Reset.Low_Duct )
   END_RUNG
   RUNG wire#w4
      Contact( "pulse_5s" )
      R_Coil( "Line_Control_DB".Line[#Alm_REQ].Messages_Reset.Low_Duct )
   END_RUNG
   // the same network as SCL:
   #_w1 := "Line_Control_DB".Line[#Alm_REQ].Messages_Reset.RT_OFF;
   IF #_w1 THEN "Line_Control_DB".Line[0].Messages_Reset.RT_OFF := TRUE; END_IF;
   IF #_w1 AND "pulse_5s" THEN "Line_Control_DB".Line[#Alm_REQ].Messages_Reset.RT_OFF := FALSE; END_IF;
   #_w2 := "Line_Control_DB".Line[#Alm_REQ].Messages_Reset.RT_ON;
   IF #_w2 THEN "Line_Control_DB".Line[0].Messages_Reset.RT_ON := TRUE; END_IF;
   IF #_w2 AND "pulse_5s" THEN "Line_Control_DB".Line[#Alm_REQ].Messages_Reset.RT_ON := FALSE; END_IF;
   #_w3 := "Line_Control_DB".Line[#Alm_REQ].Messages_Reset.Low_Conc;
   IF #_w3 THEN "Line_Control_DB".Line[0].Messages_Reset.Low_Conc := TRUE; END_IF;
   IF #_w3 AND "pulse_5s" THEN "Line_Control_DB".Line[#Alm_REQ].Messages_Reset.Low_Conc := FALSE; END_IF;
   #_w4 := "Line_Control_DB".Line[#Alm_REQ].Messages_Reset.Low_Duct;
   IF #_w4 THEN "Line_Control_DB".Line[0].Messages_Reset.Low_Duct := TRUE; END_IF;
   IF #_w4 AND "pulse_5s" THEN "Line_Control_DB".Line[#Alm_REQ].Messages_Reset.Low_Duct := FALSE; END_IF;
END_REGION

REGION Network 9: Запись данных из выбранной линии в нулевой экземпляр для отображения на дисплее
   RUNG wire#powerrail
      Move(in := "Line_Control_DB".Line[#Alm_REQ].Messages_Counter.RT_OFF, out1 => "Line_Control_DB".Line[0].Messages_Counter.RT_OFF)
      Move(in := "Line_Control_DB".Line[#Alm_REQ].Messages_Counter.RT_ON, out1 => "Line_Control_DB".Line[0].Messages_Counter.RT_ON)
      Move(in := "Line_Control_DB".Line[#Alm_REQ].Messages_Counter.Low_Conc, out1 => "Line_Control_DB".Line[0].Messages_Counter.Low_Conc)
      Move(in := "Line_Control_DB".Line[#Alm_REQ].Messages_Counter.Low_Duct, out1 => "Line_Control_DB".Line[0].Messages_Counter.Low_Duct)
   END_RUNG
   // the same network as SCL:
   "Line_Control_DB".Line[0].Messages_Counter.RT_OFF := "Line_Control_DB".Line[#Alm_REQ].Messages_Counter.RT_OFF;
   "Line_Control_DB".Line[0].Messages_Counter.RT_ON := "Line_Control_DB".Line[#Alm_REQ].Messages_Counter.RT_ON;
   "Line_Control_DB".Line[0].Messages_Counter.Low_Conc := "Line_Control_DB".Line[#Alm_REQ].Messages_Counter.Low_Conc;
   "Line_Control_DB".Line[0].Messages_Counter.Low_Duct := "Line_Control_DB".Line[#Alm_REQ].Messages_Counter.Low_Duct;
END_REGION

REGION Network 10: Чтение данных из выбранной линии в нулевой экземпляр для отображения на дисплее
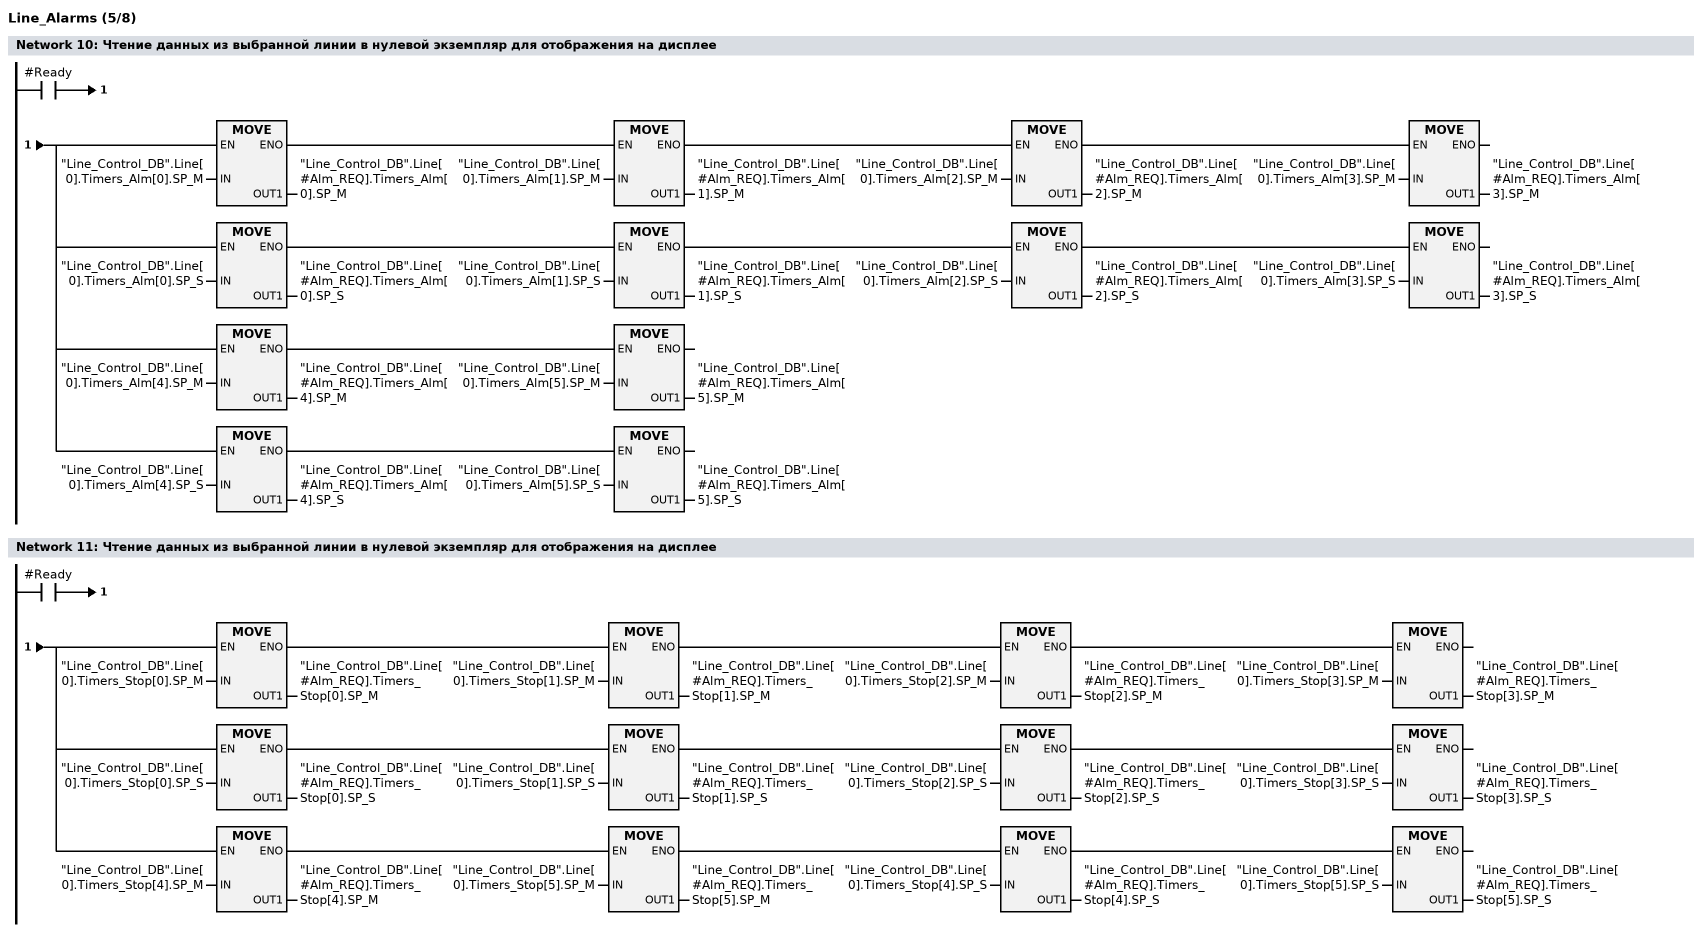
   RUNG wire#powerrail
      Contact( #Ready )
      wire#w1
      Move(in := "Line_Control_DB".Line[0].Timers_Alm[0].SP_M, out1 => "Line_Control_DB".Line[#Alm_REQ].Timers_Alm[0].SP_M)
      Move(in := "Line_Control_DB".Line[0].Timers_Alm[1].SP_M, out1 => "Line_Control_DB".Line[#Alm_REQ].Timers_Alm[1].SP_M)
      Move(in := "Line_Control_DB".Line[0].Timers_Alm[2].SP_M, out1 => "Line_Control_DB".Line[#Alm_REQ].Timers_Alm[2].SP_M)
      Move(in := "Line_Control_DB".Line[0].Timers_Alm[3].SP_M, out1 => "Line_Control_DB".Line[#Alm_REQ].Timers_Alm[3].SP_M)
   END_RUNG
   RUNG wire#w1
      Move(in := "Line_Control_DB".Line[0].Timers_Alm[0].SP_S, out1 => "Line_Control_DB".Line[#Alm_REQ].Timers_Alm[0].SP_S)
      Move(in := "Line_Control_DB".Line[0].Timers_Alm[1].SP_S, out1 => "Line_Control_DB".Line[#Alm_REQ].Timers_Alm[1].SP_S)
      Move(in := "Line_Control_DB".Line[0].Timers_Alm[2].SP_S, out1 => "Line_Control_DB".Line[#Alm_REQ].Timers_Alm[2].SP_S)
      Move(in := "Line_Control_DB".Line[0].Timers_Alm[3].SP_S, out1 => "Line_Control_DB".Line[#Alm_REQ].Timers_Alm[3].SP_S)
   END_RUNG
   RUNG wire#w1
      Move(in := "Line_Control_DB".Line[0].Timers_Alm[4].SP_M, out1 => "Line_Control_DB".Line[#Alm_REQ].Timers_Alm[4].SP_M)
      Move(in := "Line_Control_DB".Line[0].Timers_Alm[5].SP_M, out1 => "Line_Control_DB".Line[#Alm_REQ].Timers_Alm[5].SP_M)
   END_RUNG
   RUNG wire#w1
      Move(in := "Line_Control_DB".Line[0].Timers_Alm[4].SP_S, out1 => "Line_Control_DB".Line[#Alm_REQ].Timers_Alm[4].SP_S)
      Move(in := "Line_Control_DB".Line[0].Timers_Alm[5].SP_S, out1 => "Line_Control_DB".Line[#Alm_REQ].Timers_Alm[5].SP_S)
   END_RUNG
   // the same network as SCL:
   IF #Ready THEN
       "Line_Control_DB".Line[#Alm_REQ].Timers_Alm[0].SP_M := "Line_Control_DB".Line[0].Timers_Alm[0].SP_M;
       "Line_Control_DB".Line[#Alm_REQ].Timers_Alm[1].SP_M := "Line_Control_DB".Line[0].Timers_Alm[1].SP_M;
       "Line_Control_DB".Line[#Alm_REQ].Timers_Alm[2].SP_M := "Line_Control_DB".Line[0].Timers_Alm[2].SP_M;
       "Line_Control_DB".Line[#Alm_REQ].Timers_Alm[3].SP_M := "Line_Control_DB".Line[0].Timers_Alm[3].SP_M;
       "Line_Control_DB".Line[#Alm_REQ].Timers_Alm[0].SP_S := "Line_Control_DB".Line[0].Timers_Alm[0].SP_S;
       "Line_Control_DB".Line[#Alm_REQ].Timers_Alm[1].SP_S := "Line_Control_DB".Line[0].Timers_Alm[1].SP_S;
       "Line_Control_DB".Line[#Alm_REQ].Timers_Alm[2].SP_S := "Line_Control_DB".Line[0].Timers_Alm[2].SP_S;
       "Line_Control_DB".Line[#Alm_REQ].Timers_Alm[3].SP_S := "Line_Control_DB".Line[0].Timers_Alm[3].SP_S;
       "Line_Control_DB".Line[#Alm_REQ].Timers_Alm[4].SP_M := "Line_Control_DB".Line[0].Timers_Alm[4].SP_M;
       "Line_Control_DB".Line[#Alm_REQ].Timers_Alm[5].SP_M := "Line_Control_DB".Line[0].Timers_Alm[5].SP_M;
       "Line_Control_DB".Line[#Alm_REQ].Timers_Alm[4].SP_S := "Line_Control_DB".Line[0].Timers_Alm[4].SP_S;
       "Line_Control_DB".Line[#Alm_REQ].Timers_Alm[5].SP_S := "Line_Control_DB".Line[0].Timers_Alm[5].SP_S;
   END_IF;
END_REGION

REGION Network 11: Чтение данных из выбранной линии в нулевой экземпляр для отображения на дисплее
   RUNG wire#powerrail
      Contact( #Ready )
      wire#w1
      Move(in := "Line_Control_DB".Line[0].Timers_Stop[0].SP_M, out1 => "Line_Control_DB".Line[#Alm_REQ].Timers_Stop[0].SP_M)
      Move(in := "Line_Control_DB".Line[0].Timers_Stop[1].SP_M, out1 => "Line_Control_DB".Line[#Alm_REQ].Timers_Stop[1].SP_M)
      Move(in := "Line_Control_DB".Line[0].Timers_Stop[2].SP_M, out1 => "Line_Control_DB".Line[#Alm_REQ].Timers_Stop[2].SP_M)
      Move(in := "Line_Control_DB".Line[0].Timers_Stop[3].SP_M, out1 => "Line_Control_DB".Line[#Alm_REQ].Timers_Stop[3].SP_M)
   END_RUNG
   RUNG wire#w1
      Move(in := "Line_Control_DB".Line[0].Timers_Stop[0].SP_S, out1 => "Line_Control_DB".Line[#Alm_REQ].Timers_Stop[0].SP_S)
      Move(in := "Line_Control_DB".Line[0].Timers_Stop[1].SP_S, out1 => "Line_Control_DB".Line[#Alm_REQ].Timers_Stop[1].SP_S)
      Move(in := "Line_Control_DB".Line[0].Timers_Stop[2].SP_S, out1 => "Line_Control_DB".Line[#Alm_REQ].Timers_Stop[2].SP_S)
      Move(in := "Line_Control_DB".Line[0].Timers_Stop[3].SP_S, out1 => "Line_Control_DB".Line[#Alm_REQ].Timers_Stop[3].SP_S)
   END_RUNG
   RUNG wire#w1
      Move(in := "Line_Control_DB".Line[0].Timers_Stop[4].SP_M, out1 => "Line_Control_DB".Line[#Alm_REQ].Timers_Stop[4].SP_M)
      Move(in := "Line_Control_DB".Line[0].Timers_Stop[5].SP_M, out1 => "Line_Control_DB".Line[#Alm_REQ].Timers_Stop[5].SP_M)
      Move(in := "Line_Control_DB".Line[0].Timers_Stop[4].SP_S, out1 => "Line_Control_DB".Line[#Alm_REQ].Timers_Stop[4].SP_S)
      Move(in := "Line_Control_DB".Line[0].Timers_Stop[5].SP_S, out1 => "Line_Control_DB".Line[#Alm_REQ].Timers_Stop[5].SP_S)
   END_RUNG
   // the same network as SCL:
   IF #Ready THEN
       "Line_Control_DB".Line[#Alm_REQ].Timers_Stop[0].SP_M := "Line_Control_DB".Line[0].Timers_Stop[0].SP_M;
       "Line_Control_DB".Line[#Alm_REQ].Timers_Stop[1].SP_M := "Line_Control_DB".Line[0].Timers_Stop[1].SP_M;
       "Line_Control_DB".Line[#Alm_REQ].Timers_Stop[2].SP_M := "Line_Control_DB".Line[0].Timers_Stop[2].SP_M;
       "Line_Control_DB".Line[#Alm_REQ].Timers_Stop[3].SP_M := "Line_Control_DB".Line[0].Timers_Stop[3].SP_M;
       "Line_Control_DB".Line[#Alm_REQ].Timers_Stop[0].SP_S := "Line_Control_DB".Line[0].Timers_Stop[0].SP_S;
       "Line_Control_DB".Line[#Alm_REQ].Timers_Stop[1].SP_S := "Line_Control_DB".Line[0].Timers_Stop[1].SP_S;
       "Line_Control_DB".Line[#Alm_REQ].Timers_Stop[2].SP_S := "Line_Control_DB".Line[0].Timers_Stop[2].SP_S;
       "Line_Control_DB".Line[#Alm_REQ].Timers_Stop[3].SP_S := "Line_Control_DB".Line[0].Timers_Stop[3].SP_S;
       "Line_Control_DB".Line[#Alm_REQ].Timers_Stop[4].SP_M := "Line_Control_DB".Line[0].Timers_Stop[4].SP_M;
       "Line_Control_DB".Line[#Alm_REQ].Timers_Stop[5].SP_M := "Line_Control_DB".Line[0].Timers_Stop[5].SP_M;
       "Line_Control_DB".Line[#Alm_REQ].Timers_Stop[4].SP_S := "Line_Control_DB".Line[0].Timers_Stop[4].SP_S;
       "Line_Control_DB".Line[#Alm_REQ].Timers_Stop[5].SP_S := "Line_Control_DB".Line[0].Timers_Stop[5].SP_S;
   END_IF;
END_REGION

REGION Network 12: Чтение данных из выбранной линии в нулевой экземпляр для отображения на дисплее
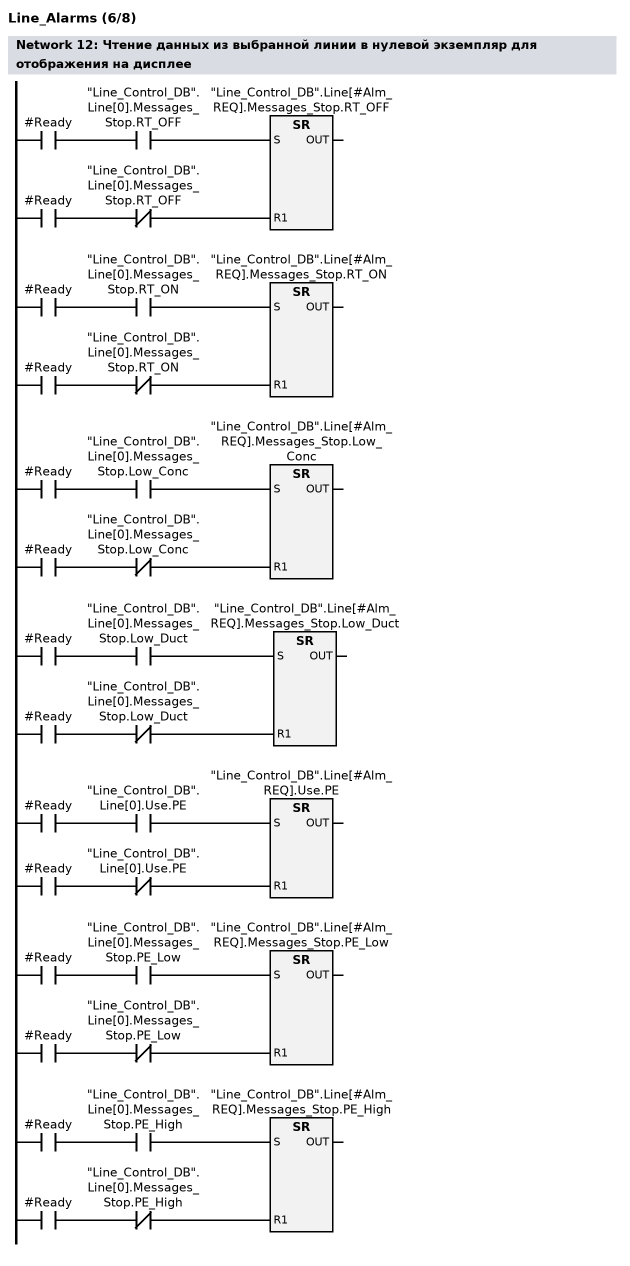
   RUNG wire#powerrail
      Contact( #Ready )
      Contact( "Line_Control_DB".Line[0].Messages_Stop.RT_OFF )
      S_SR(operand := "Line_Control_DB".Line[#Alm_REQ].Messages_Stop.RT_OFF, r1 := wire#w1)
   END_RUNG
   RUNG wire#powerrail
      Contact( #Ready )
      I_Contact( "Line_Control_DB".Line[0].Messages_Stop.RT_OFF )
   END_RUNG wire#w1
   RUNG wire#powerrail
      Contact( #Ready )
      Contact( "Line_Control_DB".Line[0].Messages_Stop.RT_ON )
      S_SR(operand := "Line_Control_DB".Line[#Alm_REQ].Messages_Stop.RT_ON, r1 := wire#w2)
   END_RUNG
   RUNG wire#powerrail
      Contact( #Ready )
      I_Contact( "Line_Control_DB".Line[0].Messages_Stop.RT_ON )
   END_RUNG wire#w2
   RUNG wire#powerrail
      Contact( #Ready )
      Contact( "Line_Control_DB".Line[0].Messages_Stop.Low_Conc )
      S_SR(operand := "Line_Control_DB".Line[#Alm_REQ].Messages_Stop.Low_Conc, r1 := wire#w3)
   END_RUNG
   RUNG wire#powerrail
      Contact( #Ready )
      I_Contact( "Line_Control_DB".Line[0].Messages_Stop.Low_Conc )
   END_RUNG wire#w3
   RUNG wire#powerrail
      Contact( #Ready )
      Contact( "Line_Control_DB".Line[0].Messages_Stop.Low_Duct )
      S_SR(operand := "Line_Control_DB".Line[#Alm_REQ].Messages_Stop.Low_Duct, r1 := wire#w4)
   END_RUNG
   RUNG wire#powerrail
      Contact( #Ready )
      I_Contact( "Line_Control_DB".Line[0].Messages_Stop.Low_Duct )
   END_RUNG wire#w4
   RUNG wire#powerrail
      Contact( #Ready )
      Contact( "Line_Control_DB".Line[0].Use.PE )
      S_SR(operand := "Line_Control_DB".Line[#Alm_REQ].Use.PE, r1 := wire#w5)
   END_RUNG
   RUNG wire#powerrail
      Contact( #Ready )
      I_Contact( "Line_Control_DB".Line[0].Use.PE )
   END_RUNG wire#w5
   RUNG wire#powerrail
      Contact( #Ready )
      Contact( "Line_Control_DB".Line[0].Messages_Stop.PE_Low )
      S_SR(operand := "Line_Control_DB".Line[#Alm_REQ].Messages_Stop.PE_Low, r1 := wire#w6)
   END_RUNG
   RUNG wire#powerrail
      Contact( #Ready )
      I_Contact( "Line_Control_DB".Line[0].Messages_Stop.PE_Low )
   END_RUNG wire#w6
   RUNG wire#powerrail
      Contact( #Ready )
      Contact( "Line_Control_DB".Line[0].Messages_Stop.PE_High )
      S_SR(operand := "Line_Control_DB".Line[#Alm_REQ].Messages_Stop.PE_High, r1 := wire#w7)
   END_RUNG
   RUNG wire#powerrail
      Contact( #Ready )
      I_Contact( "Line_Control_DB".Line[0].Messages_Stop.PE_High )
   END_RUNG wire#w7
   // the same network as SCL:
   #_w1 := #Ready AND NOT "Line_Control_DB".Line[0].Messages_Stop.RT_OFF;
   IF #Ready AND "Line_Control_DB".Line[0].Messages_Stop.RT_OFF THEN
       "Line_Control_DB".Line[#Alm_REQ].Messages_Stop.RT_OFF := TRUE;   // SR flip-flop
   END_IF;
   IF #_w1 THEN "Line_Control_DB".Line[#Alm_REQ].Messages_Stop.RT_OFF := FALSE; END_IF;
   #_w2 := #Ready AND NOT "Line_Control_DB".Line[0].Messages_Stop.RT_ON;
   IF #Ready AND "Line_Control_DB".Line[0].Messages_Stop.RT_ON THEN
       "Line_Control_DB".Line[#Alm_REQ].Messages_Stop.RT_ON := TRUE;   // SR flip-flop
   END_IF;
   IF #_w2 THEN "Line_Control_DB".Line[#Alm_REQ].Messages_Stop.RT_ON := FALSE; END_IF;
   #_w3 := #Ready AND NOT "Line_Control_DB".Line[0].Messages_Stop.Low_Conc;
   IF #Ready AND "Line_Control_DB".Line[0].Messages_Stop.Low_Conc THEN
       "Line_Control_DB".Line[#Alm_REQ].Messages_Stop.Low_Conc := TRUE;   // SR flip-flop
   END_IF;
   IF #_w3 THEN "Line_Control_DB".Line[#Alm_REQ].Messages_Stop.Low_Conc := FALSE; END_IF;
   #_w4 := #Ready AND NOT "Line_Control_DB".Line[0].Messages_Stop.Low_Duct;
   IF #Ready AND "Line_Control_DB".Line[0].Messages_Stop.Low_Duct THEN
       "Line_Control_DB".Line[#Alm_REQ].Messages_Stop.Low_Duct := TRUE;   // SR flip-flop
   END_IF;
   IF #_w4 THEN "Line_Control_DB".Line[#Alm_REQ].Messages_Stop.Low_Duct := FALSE; END_IF;
   #_w5 := #Ready AND NOT "Line_Control_DB".Line[0].Use.PE;
   IF #Ready AND "Line_Control_DB".Line[0].Use.PE THEN
       "Line_Control_DB".Line[#Alm_REQ].Use.PE := TRUE;   // SR flip-flop
   END_IF;
   IF #_w5 THEN "Line_Control_DB".Line[#Alm_REQ].Use.PE := FALSE; END_IF;
   #_w6 := #Ready AND NOT "Line_Control_DB".Line[0].Messages_Stop.PE_Low;
   IF #Ready AND "Line_Control_DB".Line[0].Messages_Stop.PE_Low THEN
       "Line_Control_DB".Line[#Alm_REQ].Messages_Stop.PE_Low := TRUE;   // SR flip-flop
   END_IF;
   IF #_w6 THEN "Line_Control_DB".Line[#Alm_REQ].Messages_Stop.PE_Low := FALSE; END_IF;
   #_w7 := #Ready AND NOT "Line_Control_DB".Line[0].Messages_Stop.PE_High;
   IF #Ready AND "Line_Control_DB".Line[0].Messages_Stop.PE_High THEN
       "Line_Control_DB".Line[#Alm_REQ].Messages_Stop.PE_High := TRUE;   // SR flip-flop
   END_IF;
   IF #_w7 THEN "Line_Control_DB".Line[#Alm_REQ].Messages_Stop.PE_High := FALSE; END_IF;
END_REGION

REGION Network 13: Чтение данных из выбранной линии в нулевой экземпляр для отображения на дисплее
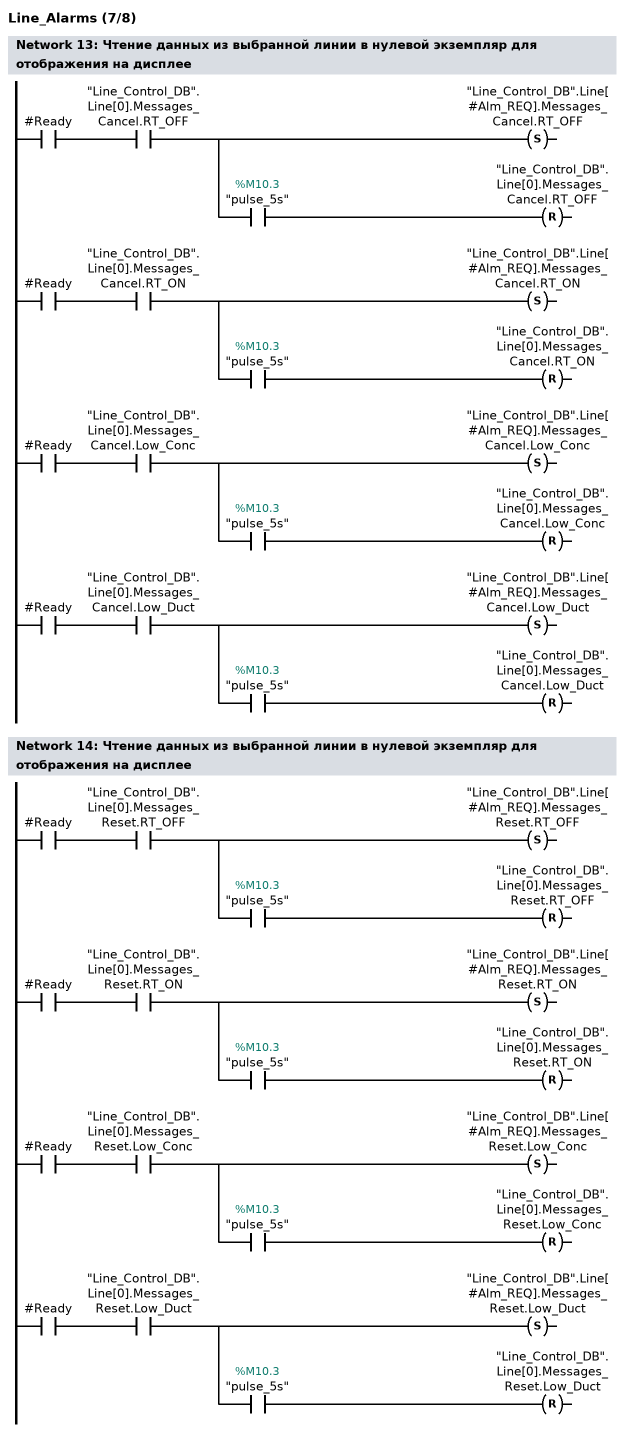
   RUNG wire#powerrail
      Contact( #Ready )
      Contact( "Line_Control_DB".Line[0].Messages_Cancel.RT_OFF )
      wire#w1
      S_Coil( "Line_Control_DB".Line[#Alm_REQ].Messages_Cancel.RT_OFF )
   END_RUNG
   RUNG wire#w1
      Contact( "pulse_5s" )
      R_Coil( "Line_Control_DB".Line[0].Messages_Cancel.RT_OFF )
   END_RUNG
   RUNG wire#powerrail
      Contact( #Ready )
      Contact( "Line_Control_DB".Line[0].Messages_Cancel.RT_ON )
      wire#w2
      S_Coil( "Line_Control_DB".Line[#Alm_REQ].Messages_Cancel.RT_ON )
   END_RUNG
   RUNG wire#w2
      Contact( "pulse_5s" )
      R_Coil( "Line_Control_DB".Line[0].Messages_Cancel.RT_ON )
   END_RUNG
   RUNG wire#powerrail
      Contact( #Ready )
      Contact( "Line_Control_DB".Line[0].Messages_Cancel.Low_Conc )
      wire#w3
      S_Coil( "Line_Control_DB".Line[#Alm_REQ].Messages_Cancel.Low_Conc )
   END_RUNG
   RUNG wire#w3
      Contact( "pulse_5s" )
      R_Coil( "Line_Control_DB".Line[0].Messages_Cancel.Low_Conc )
   END_RUNG
   RUNG wire#powerrail
      Contact( #Ready )
      Contact( "Line_Control_DB".Line[0].Messages_Cancel.Low_Duct )
      wire#w4
      S_Coil( "Line_Control_DB".Line[#Alm_REQ].Messages_Cancel.Low_Duct )
   END_RUNG
   RUNG wire#w4
      Contact( "pulse_5s" )
      R_Coil( "Line_Control_DB".Line[0].Messages_Cancel.Low_Duct )
   END_RUNG
   // the same network as SCL:
   #_w1 := #Ready AND "Line_Control_DB".Line[0].Messages_Cancel.RT_OFF;
   IF #_w1 THEN "Line_Control_DB".Line[#Alm_REQ].Messages_Cancel.RT_OFF := TRUE; END_IF;
   IF #_w1 AND "pulse_5s" THEN "Line_Control_DB".Line[0].Messages_Cancel.RT_OFF := FALSE; END_IF;
   #_w2 := #Ready AND "Line_Control_DB".Line[0].Messages_Cancel.RT_ON;
   IF #_w2 THEN "Line_Control_DB".Line[#Alm_REQ].Messages_Cancel.RT_ON := TRUE; END_IF;
   IF #_w2 AND "pulse_5s" THEN "Line_Control_DB".Line[0].Messages_Cancel.RT_ON := FALSE; END_IF;
   #_w3 := #Ready AND "Line_Control_DB".Line[0].Messages_Cancel.Low_Conc;
   IF #_w3 THEN "Line_Control_DB".Line[#Alm_REQ].Messages_Cancel.Low_Conc := TRUE; END_IF;
   IF #_w3 AND "pulse_5s" THEN "Line_Control_DB".Line[0].Messages_Cancel.Low_Conc := FALSE; END_IF;
   #_w4 := #Ready AND "Line_Control_DB".Line[0].Messages_Cancel.Low_Duct;
   IF #_w4 THEN "Line_Control_DB".Line[#Alm_REQ].Messages_Cancel.Low_Duct := TRUE; END_IF;
   IF #_w4 AND "pulse_5s" THEN "Line_Control_DB".Line[0].Messages_Cancel.Low_Duct := FALSE; END_IF;
END_REGION

REGION Network 14: Чтение данных из выбранной линии в нулевой экземпляр для отображения на дисплее
   RUNG wire#powerrail
      Contact( #Ready )
      Contact( "Line_Control_DB".Line[0].Messages_Reset.RT_OFF )
      wire#w1
      S_Coil( "Line_Control_DB".Line[#Alm_REQ].Messages_Reset.RT_OFF )
   END_RUNG
   RUNG wire#w1
      Contact( "pulse_5s" )
      R_Coil( "Line_Control_DB".Line[0].Messages_Reset.RT_OFF )
   END_RUNG
   RUNG wire#powerrail
      Contact( #Ready )
      Contact( "Line_Control_DB".Line[0].Messages_Reset.RT_ON )
      wire#w2
      S_Coil( "Line_Control_DB".Line[#Alm_REQ].Messages_Reset.RT_ON )
   END_RUNG
   RUNG wire#w2
      Contact( "pulse_5s" )
      R_Coil( "Line_Control_DB".Line[0].Messages_Reset.RT_ON )
   END_RUNG
   RUNG wire#powerrail
      Contact( #Ready )
      Contact( "Line_Control_DB".Line[0].Messages_Reset.Low_Conc )
      wire#w3
      S_Coil( "Line_Control_DB".Line[#Alm_REQ].Messages_Reset.Low_Conc )
   END_RUNG
   RUNG wire#w3
      Contact( "pulse_5s" )
      R_Coil( "Line_Control_DB".Line[0].Messages_Reset.Low_Conc )
   END_RUNG
   RUNG wire#powerrail
      Contact( #Ready )
      Contact( "Line_Control_DB".Line[0].Messages_Reset.Low_Duct )
      wire#w4
      S_Coil( "Line_Control_DB".Line[#Alm_REQ].Messages_Reset.Low_Duct )
   END_RUNG
   RUNG wire#w4
      Contact( "pulse_5s" )
      R_Coil( "Line_Control_DB".Line[0].Messages_Reset.Low_Duct )
   END_RUNG
   // the same network as SCL:
   #_w1 := #Ready AND "Line_Control_DB".Line[0].Messages_Reset.RT_OFF;
   IF #_w1 THEN "Line_Control_DB".Line[#Alm_REQ].Messages_Reset.RT_OFF := TRUE; END_IF;
   IF #_w1 AND "pulse_5s" THEN "Line_Control_DB".Line[0].Messages_Reset.RT_OFF := FALSE; END_IF;
   #_w2 := #Ready AND "Line_Control_DB".Line[0].Messages_Reset.RT_ON;
   IF #_w2 THEN "Line_Control_DB".Line[#Alm_REQ].Messages_Reset.RT_ON := TRUE; END_IF;
   IF #_w2 AND "pulse_5s" THEN "Line_Control_DB".Line[0].Messages_Reset.RT_ON := FALSE; END_IF;
   #_w3 := #Ready AND "Line_Control_DB".Line[0].Messages_Reset.Low_Conc;
   IF #_w3 THEN "Line_Control_DB".Line[#Alm_REQ].Messages_Reset.Low_Conc := TRUE; END_IF;
   IF #_w3 AND "pulse_5s" THEN "Line_Control_DB".Line[0].Messages_Reset.Low_Conc := FALSE; END_IF;
   #_w4 := #Ready AND "Line_Control_DB".Line[0].Messages_Reset.Low_Duct;
   IF #_w4 THEN "Line_Control_DB".Line[#Alm_REQ].Messages_Reset.Low_Duct := TRUE; END_IF;
   IF #_w4 AND "pulse_5s" THEN "Line_Control_DB".Line[0].Messages_Reset.Low_Duct := FALSE; END_IF;
END_REGION

REGION Network 15: Чтение данных из выбранной линии в нулевой экземпляр для отображения на дисплее
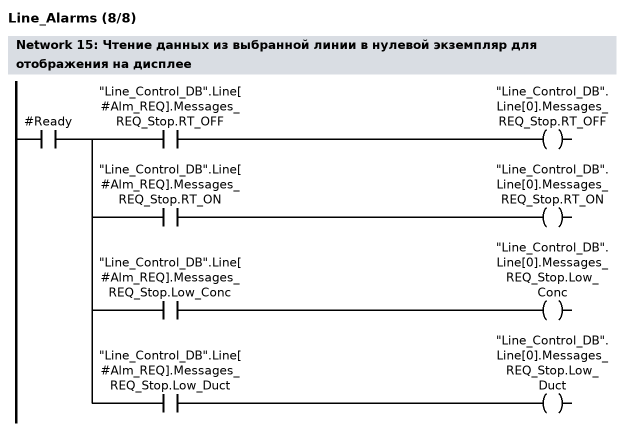
   RUNG wire#powerrail
      Contact( #Ready )
      wire#w1
      Contact( "Line_Control_DB".Line[#Alm_REQ].Messages_REQ_Stop.RT_OFF )
      Coil( "Line_Control_DB".Line[0].Messages_REQ_Stop.RT_OFF )
   END_RUNG
   RUNG wire#w1
      Contact( "Line_Control_DB".Line[#Alm_REQ].Messages_REQ_Stop.RT_ON )
      Coil( "Line_Control_DB".Line[0].Messages_REQ_Stop.RT_ON )
   END_RUNG
   RUNG wire#w1
      Contact( "Line_Control_DB".Line[#Alm_REQ].Messages_REQ_Stop.Low_Conc )
      Coil( "Line_Control_DB".Line[0].Messages_REQ_Stop.Low_Conc )
   END_RUNG
   RUNG wire#w1
      Contact( "Line_Control_DB".Line[#Alm_REQ].Messages_REQ_Stop.Low_Duct )
      Coil( "Line_Control_DB".Line[0].Messages_REQ_Stop.Low_Duct )
   END_RUNG
   // the same network as SCL:
   "Line_Control_DB".Line[0].Messages_REQ_Stop.RT_OFF := #Ready AND "Line_Control_DB".Line[#Alm_REQ].Messages_REQ_Stop.RT_OFF;
   "Line_Control_DB".Line[0].Messages_REQ_Stop.RT_ON := #Ready AND "Line_Control_DB".Line[#Alm_REQ].Messages_REQ_Stop.RT_ON;
   "Line_Control_DB".Line[0].Messages_REQ_Stop.Low_Conc := #Ready AND "Line_Control_DB".Line[#Alm_REQ].Messages_REQ_Stop.Low_Conc;
   "Line_Control_DB".Line[0].Messages_REQ_Stop.Low_Duct := #Ready AND "Line_Control_DB".Line[#Alm_REQ].Messages_REQ_Stop.Low_Duct;
END_REGION
END_FUNCTION

FUNCTION_BLOCK "Block_Line"   // FB12, LAD
{ S7_Optimized_Access := 'TRUE' }
VERSION : 0.1
// stored: AutoNumber true, IsIECCheckEnabled false, IsRetainMemResEnabled false, MemoryReserve 100, SetENOAutomatically false, UDAEnableTagReadback false
   VAR_INPUT
      Flow : Real;   // Расходомер принимающей трубы
      SP_C : Real := 0.01;   // Уставка дозации, % масс, 0.05-1
      PE : Real;   // Датчик давления
      ALLS : Bool;   // Авариййный нижний уровень бака
      RT : Bool;   // Ротаметр
      RM : Bool;   // Датчик протока вместо расходомера
      KC_ON : Bool;   // Клапан открыт
      PE_LLS : Bool;
      PE_HHS : Bool;
   END_VAR
   VAR_OUTPUT
      KC_CMD : Bool;   // Открытие клапана
   END_VAR
   VAR_IN_OUT
      Report_H : "Line_Report";   // Разовый отчёт
   END_VAR
   VAR RETAIN
      LINE_NUMBER : Int;   // номер линии
   END_VAR
   VAR
      Start : Bool;   // Запуск линии
      Main_ON : Bool;   // Команда основного насоса
      Reserv_ON : Bool;   // Команда резервного насоса
   END_VAR
   VAR RETAIN
      Hand { S7_SetPoint := 'True'} : Bool;   // 1 - Задание скорости насосов в ручном режиме
      Choice_Tank : Bool;   // 0 - основной танк, 1 - резервный
      SP_Source { S7_SetPoint := 'True'} : Bool;   // 0 - по формуле расчета, 1 - равен входу Flow
      PID_Not_Use { S7_SetPoint := 'True'} : Bool;   // Использовать ПИД (0 - использовать, 1 - не использовать)
      Mode { S7_SetPoint := 'True'} : Bool;   // 0 - без разбаления, 1 - с разбавлением
      Mode_Local : Bool;   // Режим: 0 - местный, 1 - локальный
   END_VAR
   VAR
      Res_CMD : Bool;   // Команда ротации по наработке
      Res_ANY : Bool;   // Первый насос в резерве
      No_Water : Bool;   // Авария "Нет продукта" HMI
      Dry_Run : Bool;   // Авария "Нет протока, сухой ход" HMI
      Pump_Main_Alarm : Bool;   // Выходной сигнал аварии насоса 1
      Pump_Reserv_Alarm : Bool;   // Выходной сигнал аварии насоса 2
      Main_Line_Ok : Bool := true;   // Готовность основной линии
      Low_Stop : Bool;   // Остановка по низкому протоку
      RM_1_Alarm : Bool;   // Авария основного расходомера
      RM_2_Alarm : Bool;   // Авария дополнительного расходомера
   END_VAR
   VAR RETAIN
      RM_1_Report_DI { S7_SetPoint := 'True'} : Bool;   // Использовать импусльный сигнал для отчётов
      RM_2_Report_DI { S7_SetPoint := 'True'} : Bool;   // Использовать импусльный сигнал для отчётов
      RM_Weight { S7_SetPoint := 'True'} : Real := 1.0;   // Вес импульса
   END_VAR
   VAR
      Status_Main : Int;   // Статус основного насоса
      Status_Reserv : Int;   // Статус резервного насоса
      Events : Word;   // События линии
      SP_A : Real;   // Уставка авторежима
   END_VAR
   VAR RETAIN
      SP_M { S7_SetPoint := 'True'} : Real;   // Уставка ручного режима
      SP_min { S7_SetPoint := 'True'} : Real := 10.0;   // Минимальная скорость насоса
      SP_max { S7_SetPoint := 'True'} : Real := 1000.0;   // Максимальная скорость насоса
      PE_min { S7_SetPoint := 'True'} : Real := 0.15;   // Низкое давление в линии
      PE_max { S7_SetPoint := 'True'} : Real := 2.5;   // Высокое давление в линии
   END_VAR
   VAR
      Pump_SP : Real;   // Актуальная скорость насоса
   END_VAR
   VAR RETAIN
      D { S7_SetPoint := 'True'} : Real;   // Уставка дозы
      D_Num : Real;   // Количество замерок дозы
      D_Sum : Real;   // Общаяя сумма дозы
   END_VAR
   VAR
      C : Real;   // Рабочие данные о концентрации
   END_VAR
   VAR RETAIN
      C_Tank { S7_SetPoint := 'True'} : Real;   // Концентрация в резервном баке
   END_VAR
   VAR
      Flow_Line : Real;   // Расходомер, используемый в данный момент
      Flow_s { ExternalAccessible := 'False'; ExternalVisible := 'False'; ExternalWritable := 'False'} : Real;   // Переведенный в секунды
      Alarm_SP : Real;   // Аварийный коэфф соотношение уставки к реальной скорости насоса
   END_VAR
   VAR RETAIN
      Low_Flow { S7_SetPoint := 'True'} : Real;   // Низкий проток в основной линии
      Res_Main : Real;   // Наработка основного насоса
      Res_Reserv : Real;   // Наработка резревного насоса
      Res_SP { S7_SetPoint := 'True'} : Real;   // Уставка переключения по наработке
   END_VAR
   VAR
      Last_D : Real;   // Предъдущее значение дозы
      Last_SP : Real;   // Предъдущее значение расхода
   END_VAR
   VAR RETAIN
      Use : Struct   // Конфигурация
         RT { S7_SetPoint := 'True'} : Bool;   // Использование ротаметра
         RM { S7_SetPoint := 'True'} : Bool;   // Использование датчика протока вместо расходомера
         SP { S7_SetPoint := 'True'} : Bool := true;   // Использовать аналоговое регулирование
         Flow { S7_SetPoint := 'True'} : Bool := true;   // Использовать контрольный расходомер
         Res { S7_SetPoint := 'True'} : Bool;   // Использовать переключение по наработке
         DME { S7_SetPoint := 'True'} : Bool;   // Мембранные насосы
         PE { S7_SetPoint := 'True'} : Bool;
      END_STRUCT;
   END_VAR
   VAR
      Messages : Struct   // - Аварийные сообщения
         Low_Duct : Bool;   // Авария - низкий проток
         Low_Conc : Bool;   // Авария - низкая концентрация
         RT_ON : Bool;   // Авария - нет протока воды на ротаметре
         RT_OFF : Bool;   // Авария - поток воды не пропал на ротаметре
         RM_Error : Bool;   // Авария - неисправен расходомер
         PE_Low : Bool;   // Авария - низкое давление в линии
         PE_High : Bool;   // Авария - высокое давление в линии
         Alarm : Word;   // Слово аварий для панели
      END_STRUCT;
      Messages_Cancel : Struct   // - Отмена остановки
         Low_Duct : Bool;   // Авария - низкий проток
         Low_Conc : Bool;   // Авария - низкая концентрация
         RT_ON : Bool;   // Авария - нет протока воды на ротаметре
         RT_OFF : Bool;   // Авария - поток воды не пропал на ротаметре
         PE_Low : Bool;   // Авария - низкое давление в линии
         PE_High : Bool;   // Авария - высокое давление в линии
      END_STRUCT;
      Messages_Stop : Struct   // - Остановка по аварии
         Low_Duct : Bool;   // Авария - низкий проток
         Low_Conc : Bool;   // Авария - низкая концентрация
         RT_ON : Bool;   // Авария - нет протока воды на ротаметре
         RT_OFF : Bool;   // Авария - поток воды не пропал на ротаметре
         PE_Low : Bool;   // Авария - низкое давление в линии
         PE_High : Bool;   // Авария - высокое давление в линии
      END_STRUCT;
      Messages_Counter : Struct   // - Счётчик аварийных срабатываний
         Low_Duct : Int;   // Авария - низкий проток
         Low_Conc : Int;   // Авария - низкая концентрация
         RT_ON : Int;   // Авария - нет протока воды на ротаметре
         RT_OFF : Int;   // Авария - поток воды не пропал на ротаметре
         PE_Low : Int;   // Авария - низкое давление в линии
         PE_High : Int;   // Авария - высокое давление в линии
      END_STRUCT;
      Messages_Reset : Struct   // - Сброс счётчика
         Low_Duct : Bool;   // Авария - низкий проток
         Low_Conc : Bool;   // Авария - низкая концентрация
         RT_ON : Bool;   // Авария - нет протока воды на ротаметре
         RT_OFF : Bool;   // Авария - поток воды не пропал на ротаметре
         PE_Low : Bool;   // Авария - низкое давление в линии
         PE_High : Bool;   // Авария - высокое давление в линии
      END_STRUCT;
      Messages_REQ_Stop : Struct   // - Запрос остановки по аварии
         Low_Duct : Bool;   // Авария - низкий проток
         Low_Conc : Bool;   // Авария - низкая концентрация
         RT_ON : Bool;   // Авария - нет протока воды на ротаметре
         RT_OFF : Bool;   // Авария - поток воды не пропал на ротаметре
         PE_Low : Bool;   // Авария - низкое давление в линии
         PE_High : Bool;   // Авария - высокое давление в линии
      END_STRUCT;
      Timers_Stop : Array[0..5] of "Time_M";   // Таймеры останова
      Timers_Alm : Array[0..5] of "Time_M";   // Таймеры аварий
      T_Main_Alarm : "Time_M";   // Авария основного насоса по датчику протока
      T_Reserv_Alarm : "Time_M";   // Авария резервного насоса по датчику протока
      T_Main_Line_Ok : "Time_M";   // Таймер готовности основной линии
      T_No_Water : "Time_M";   // Нет продукта в баке
      T_Dry_Run : "Time_M";   // Нет протока в линии
      pos : Array[0..15] of Bool;   // Вспомогательные переменные
      PID { S7_SetPoint := 'True'} : "PID_ex";
      FlowMeter_1 { S7_SetPoint := 'True'} : "DRV_Flow_old";   // Расход 1
      FlowMeter_2 { S7_SetPoint := 'True'} : "DRV_Flow_old";   // Расход 2
   END_VAR
   VAR_TEMP
      ev : Bool;
      x : Real;
   END_VAR
   VAR CONSTANT
      "1s" : Real := 0.00028;
      "1m" : Real := 0.017;
   END_VAR
   // // Report_H.Res_1 : Резерв 1
   // // Report_H.Res_2 : Резерв 2
   VAR_TEMP   // added for the SCL form of the ladder/FBD networks
      _w1 : Bool;
      _w2 : Bool;
      _w3 : Bool;
      _w4 : Bool;
      _w5 : Bool;
      _w6 : Bool;
      _w7 : Bool;
      _w8 : Bool;
      _w9 : Bool;
      _w10 : Bool;
      _w11 : Bool;
      _w12 : Bool;
      _w13 : Bool;
      _w14 : Bool;
   END_VAR
BEGIN

REGION Network 1: Режим: 0 - местный, 1 - локальный
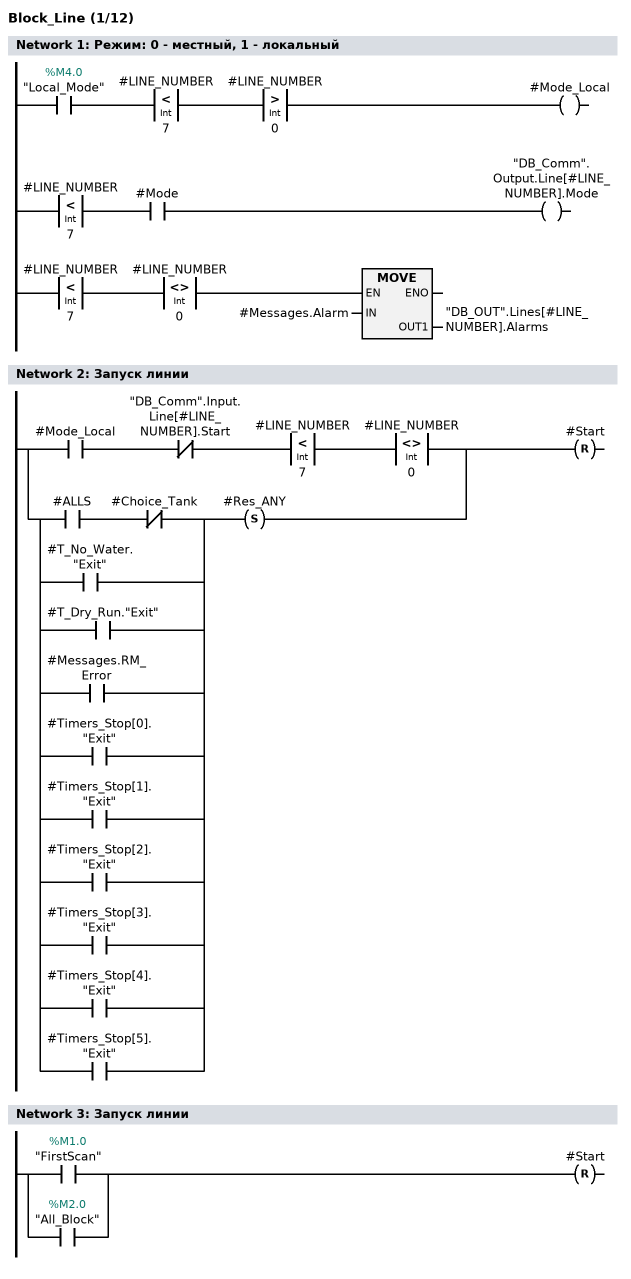
   RUNG wire#powerrail
      Contact( "Local_Mode" )
      { S7_Templates := "SrcType := Int" } LT_Contact(in1 := #LINE_NUMBER, in2 := 7)
      { S7_Templates := "SrcType := Int" } GT_Contact(in1 := #LINE_NUMBER, in2 := 0)
      Coil( #Mode_Local )
   END_RUNG
   RUNG wire#powerrail
      { S7_Templates := "SrcType := Int" } LT_Contact(in1 := #LINE_NUMBER, in2 := 7)
      Contact( #Mode )
      Coil( "DB_Comm".Output.Line[#LINE_NUMBER].Mode )
   END_RUNG
   RUNG wire#powerrail
      { S7_Templates := "SrcType := Int" } LT_Contact(in1 := #LINE_NUMBER, in2 := 7)
      { S7_Templates := "SrcType := Int" } NE_Contact(in1 := #LINE_NUMBER, in2 := 0)
      Move(in := #Messages.Alarm, out1 => "DB_OUT".Lines[#LINE_NUMBER].Alarms)
   END_RUNG
   // the same network as SCL:
   #Mode_Local := "Local_Mode" AND (#LINE_NUMBER < 7) AND (#LINE_NUMBER > 0);
   "DB_Comm".Output.Line[#LINE_NUMBER].Mode := (#LINE_NUMBER < 7) AND #Mode;
   IF (#LINE_NUMBER < 7) AND (#LINE_NUMBER <> 0) THEN
       "DB_OUT".Lines[#LINE_NUMBER].Alarms := #Messages.Alarm;
   END_IF;
END_REGION

REGION Network 2: Запуск линии
   RUNG wire#powerrail
      Contact( #Mode_Local )
      I_Contact( "DB_Comm".Input.Line[#LINE_NUMBER].Start )
      { S7_Templates := "SrcType := Int" } LT_Contact(in1 := #LINE_NUMBER, in2 := 7)
      { S7_Templates := "SrcType := Int" } NE_Contact(in1 := #LINE_NUMBER, in2 := 0)
      wire#w1
      R_Coil( #Start )
   END_RUNG
   RUNG wire#powerrail
      Contact( #ALLS )
      I_Contact( #Choice_Tank )
      wire#w2
      S_Coil( #Res_ANY )
   END_RUNG wire#w1
   RUNG wire#powerrail
      Contact( #T_No_Water."Exit" )
   END_RUNG wire#w2
   RUNG wire#powerrail
      Contact( #T_Dry_Run."Exit" )
   END_RUNG wire#w2
   RUNG wire#powerrail
      Contact( #Messages.RM_Error )
   END_RUNG wire#w2
   RUNG wire#powerrail
      Contact( #Timers_Stop[0]."Exit" )
   END_RUNG wire#w2
   RUNG wire#powerrail
      Contact( #Timers_Stop[1]."Exit" )
   END_RUNG wire#w2
   RUNG wire#powerrail
      Contact( #Timers_Stop[2]."Exit" )
   END_RUNG wire#w2
   RUNG wire#powerrail
      Contact( #Timers_Stop[3]."Exit" )
   END_RUNG wire#w2
   RUNG wire#powerrail
      Contact( #Timers_Stop[4]."Exit" )
   END_RUNG wire#w2
   RUNG wire#powerrail
      Contact( #Timers_Stop[5]."Exit" )
   END_RUNG wire#w2
   // the same network as SCL:
   #_w1 := (#ALLS AND NOT #Choice_Tank) OR #T_No_Water."Exit" OR #T_Dry_Run."Exit" OR #Messages.RM_Error OR #Timers_Stop[0]."Exit" OR #Timers_Stop[1]."Exit" OR #Timers_Stop[2]."Exit" OR #Timers_Stop[3]."Exit" OR #Timers_Stop[4]."Exit" OR #Timers_Stop[5]."Exit";
   IF #_w1 THEN #Res_ANY := TRUE; END_IF;
   IF (#Mode_Local AND NOT "DB_Comm".Input.Line[#LINE_NUMBER].Start AND (#LINE_NUMBER < 7) AND (#LINE_NUMBER <> 0)) OR #_w1 THEN
       #Start := FALSE;
   END_IF;
END_REGION

REGION Network 3: Запуск линии
   RUNG wire#powerrail
      Contact( "FirstScan" )
      wire#w1
      R_Coil( #Start )
   END_RUNG
   RUNG wire#powerrail
      Contact( "All_Block" )
   END_RUNG wire#w1
   // the same network as SCL:
   IF "FirstScan" OR "All_Block" THEN #Start := FALSE; END_IF;
END_REGION

